LIN {X 0,Y 260.818,Z 776.411,A -85,B 0,C 180,E1 -18784.461,E2 -18784.461} C_VEL
LIN {X 0,Y 257.171,Z 786.546,A -85,B 0,C 180,E1 -18786.657,E2 -18786.657} C_VEL
LIN {X 0,Y 253.713,Z 796.339,A -85,B 0,C 180,E1 -18789.319,E2 -18789.319} C_VEL
LIN {X 0,Y 251.091,Z 804.227,A -85,B 0,C 180,E1 -18792.069,E2 -18792.069} C_VEL
LIN {X 0,Y 249.103,Z 811.376,A -85,B 0,C 180,E1 -18795.292,E2 -18795.292} C_VEL
LIN {X 0,Y 248.205,Z 815.496,A -85,B 0,C 180,E1 -18797.74,E2 -18797.74} C_VEL
LIN {X 0,Y 247.91,Z 818.682,A -85,B 0,C 180,E1 -18800.208,E2 -18800.208} C_VEL
LIN {X 0,Y 248.066,Z 820.87,A -85,B 0,C 180,E1 -18802.569,E2 -18802.569} C_VEL
LIN {X 0,Y 248.583,Z 822.288,A -85,B 0,C 180,E1 -18805.135,E2 -18805.135} C_VEL
LIN {X 0,Y 248.948,Z 822.609,A -85,B 0,C 180,E1 -18806.764,E2 -18806.764} C_VEL
LIN {X 0,Y 249.746,Z 822.308,A -85,B 0,C 180,E1 -18809.396,E2 -18809.396} C_VEL
LIN {X 0,Y 249.833,Z 822.747,A -85,B 0,C 180,E1 -18810.001,E2 -18810.001} C_VEL
LIN {X 0,Y 249.274,Z 823.471,A -85,B 0,C 180,E1 -18811.617,E2 -18811.617} C_VEL
LIN {X 0,Y 248.833,Z 823.769,A -85,B 0,C 180,E1 -18813.239,E2 -18813.239} C_VEL
LIN {X 0,Y 248.449,Z 823.635,A -85,B 0,C 180,E1 -18814.869,E2 -18814.869} C_VEL
LIN {X 0,Y 247.848,Z 822.097,A -85,B 0,C 180,E1 -18818.152,E2 -18818.152} C_VEL
LIN {X 0,Y 247.929,Z 818.939,A -85,B 0,C 180,E1 -18821.446,E2 -18821.446} C_VEL
LIN {X 0,Y 248.989,Z 814.223,A -85,B 0,C 180,E1 -18824.717,E2 -18824.717} C_VEL
LIN {X 0,Y 250.924,Z 807.901,A -85,B 0,C 180,E1 -18827.945,E2 -18827.945} C_VEL
LIN {X 0,Y 253.773,Z 800.921,A -85,B 0,C 180,E1 -18830.678,E2 -18830.678} C_VEL
LIN {X 0,Y 257.433,Z 792.435,A -85,B 0,C 180,E1 -18833.32,E2 -18833.32} C_VEL
LIN {X 0,Y 261.134,Z 783.798,A -85,B 0,C 180,E1 -18835.507,E2 -18835.507} C_VEL
LIN {X 0,Y 266.249,Z 771.804,A -85,B 0,C 180,E1 -18837.94,E2 -18837.94} C_VEL
LIN {X 0,Y 271.015,Z 760.595,A -85,B 0,C 180,E1 -18839.733,E2 -18839.733} C_VEL
LIN {X 0,Y 276.161,Z 747.47,A -85,B 0,C 180,E1 -18841.447,E2 -18841.447} C_VEL
LIN {X 0,Y 281.786,Z 731.575,A -85,B 0,C 180,E1 -18843.065,E2 -18843.065} C_VEL
LIN {X 0,Y 286.827,Z 715.559,A -85,B 0,C 180,E1 -18844.303,E2 -18844.303} C_VEL
LIN {X 0,Y 291.383,Z 697.801,A -85,B 0,C 180,E1 -18845.372,E2 -18845.372} C_VEL
LIN {X 0,Y 293.955,Z 682.068,A -85,B 0,C 180,E1 -18846.336,E2 -18846.336} C_VEL
LIN {X 0,Y 295.389,Z 669.131,A -85,B 0,C 180,E1 -18847.143,E2 -18847.143} C_VEL
LIN {X 0,Y 296.48,Z 656.031,A -85,B 0,C 180,E1 -18848.176,E2 -18848.176} C_VEL
LIN {X 0,Y 297.436,Z 642.354,A -85,B 0,C 180,E1 -18849.532,E2 -18849.532} C_VEL
LIN {X 0,Y 298.39,Z 628.951,A -85,B 0,C 180,E1 -18851.163,E2 -18851.163} C_VEL
LIN {X 0,Y 298.557,Z 626.848,A -85,B 0,C 180,E1 -18851.458,E2 -18851.458} C_VEL
LIN {X 0,Y 297.497,Z 623.568,A -85,B 0,C 180,E1 -18853.968,E2 -18853.968} C_VEL
LIN {X 0,Y 297.34,Z 623.4,A -85,B 0,C 180,E1 -18856.728,E2 -18856.728} C_VEL
LIN {X 0,Y 297.736,Z 623.726,A -85,B 0,C 180,E1 -18857.889,E2 -18857.889} C_VEL
LIN {X 0,Y 299.108,Z 626.961,A -85,B 0,C 180,E1 -18860.284,E2 -18860.284} C_VEL
LIN {X 0,Y 300.421,Z 629.677,A -85,B 0,C 180,E1 -18861.677,E2 -18861.677} C_VEL
LIN {X 0,Y 301.995,Z 633.313,A -85,B 0,C 180,E1 -18863.024,E2 -18863.024} C_VEL
LIN {X 0,Y 299.757,Z 652.581,A -85,B 0,C 180,E1 -18864.07,E2 -18864.07} C_VEL
LIN {X 0,Y 297.384,Z 666.673,A -85,B 0,C 180,E1 -18865.096,E2 -18865.096} C_VEL
LIN {X 0,Y 294.073,Z 681.241,A -85,B 0,C 180,E1 -18866.45,E2 -18866.45} C_VEL
LIN {X 0,Y 290.628,Z 693.312,A -85,B 0,C 180,E1 -18867.858,E2 -18867.858} C_VEL
LIN {X 0,Y 286.356,Z 705.963,A -85,B 0,C 180,E1 -18869.684,E2 -18869.684} C_VEL
LIN {X 0,Y 282.513,Z 715.583,A -85,B 0,C 180,E1 -18871.387,E2 -18871.387} C_VEL
LIN {X 0,Y 278.319,Z 724.834,A -85,B 0,C 180,E1 -18873.37,E2 -18873.37} C_VEL
LIN {X 0,Y 273.752,Z 733.753,A -85,B 0,C 180,E1 -18875.746,E2 -18875.746} C_VEL
LIN {X 0,Y 268.985,Z 741.99,A -85,B 0,C 180,E1 -18878.543,E2 -18878.543} C_VEL
LIN {X 0,Y 264.72,Z 748.465,A -85,B 0,C 180,E1 -18881.422,E2 -18881.422} C_VEL
LIN {X 0,Y 260.983,Z 753.365,A -85,B 0,C 180,E1 -18884.377,E2 -18884.377} C_VEL
LIN {X 0,Y 257.686,Z 756.898,A -85,B 0,C 180,E1 -18887.397,E2 -18887.397} C_VEL
LIN {X 0,Y 255.181,Z 759.04,A -85,B 0,C 180,E1 -18890.488,E2 -18890.488} C_VEL
LIN {X 0,Y 253.034,Z 760.013,A -85,B 0,C 180,E1 -18893.621,E2 -18893.621} C_VEL
LIN {X 0,Y 251.501,Z 759.716,A -85,B 0,C 180,E1 -18896.795,E2 -18896.795} C_VEL
LIN {X 0,Y 250.423,Z 758.19,A -85,B 0,C 180,E1 -18899.999,E2 -18899.999} C_VEL
LIN {X 0,Y 249.712,Z 755.413,A -85,B 0,C 180,E1 -18903.226,E2 -18903.226} C_VEL
LIN {X 0,Y 249.459,Z 751.304,A -85,B 0,C 180,E1 -18906.47,E2 -18906.47} C_VEL
LIN {X 0,Y 249.698,Z 745.77,A -85,B 0,C 180,E1 -18909.722,E2 -18909.722} C_VEL
LIN {X 0,Y 250.129,Z 738.659,A -85,B 0,C 180,E1 -18912.989,E2 -18912.989} C_VEL
LIN {X 0,Y 250.911,Z 730.916,A -85,B 0,C 180,E1 -18915.848,E2 -18915.848} C_VEL
LIN {X 0,Y 252.025,Z 721.082,A -85,B 0,C 180,E1 -18918.823,E2 -18918.823} C_VEL
LIN {X 0,Y 253.137,Z 711.784,A -85,B 0,C 180,E1 -18921.156,E2 -18921.156} C_VEL
LIN {X 0,Y 254.594,Z 700.217,A -85,B 0,C 180,E1 -18923.594,E2 -18923.594} C_VEL
LIN {X 0,Y 256.131,Z 687.264,A -85,B 0,C 180,E1 -18925.84,E2 -18925.84} C_VEL
LIN {X 0,Y 257.565,Z 674.72,A -85,B 0,C 180,E1 -18927.636,E2 -18927.636} C_VEL
LIN {X 0,Y 258.908,Z 660.999,A -85,B 0,C 180,E1 -18929.248,E2 -18929.248} C_VEL
LIN {X 0,Y 260.031,Z 646.822,A -85,B 0,C 180,E1 -18930.585,E2 -18930.585} C_VEL
LIN {X 0,Y 261.021,Z 631.089,A -85,B 0,C 180,E1 -18931.727,E2 -18931.727} C_VEL
LIN {X 0,Y 261.687,Z 615.325,A -85,B 0,C 180,E1 -18932.546,E2 -18932.546} C_VEL
LIN {X 0,Y 261.742,Z 605.267,A -85,B 0,C 180,E1 -18932.982,E2 -18932.982} C_VEL
LIN {X 0,Y 249.083,Z 569.455,A -85,B 0,C 180,E1 -18935.438,E2 -18935.438} C_VEL
LIN {X 0,Y 249.029,Z 569.466,A -85,B 0,C 180,E1 -18938.379,E2 -18938.379} C_VEL
LIN {X 0,Y 249.01,Z 569.466,A -85,B 0,C 180,E1 -18942.791,E2 -18942.791} C_VEL
LIN {X 0,Y 249.02,Z 569.462,A -85,B 0,C 180,E1 -18947.362,E2 -18947.362} C_VEL
LIN {X 0,Y 249.04,Z 569.461,A -85,B 0,C 180,E1 -18951.621,E2 -18951.621} C_VEL
LIN {X 0,Y 249.061,Z 569.458,A -85,B 0,C 180,E1 -18955.641,E2 -18955.641} C_VEL
LIN {X 0,Y 249.047,Z 569.459,A -85,B 0,C 180,E1 -18959.471,E2 -18959.471} C_VEL
LIN {X 0,Y 249.071,Z 569.458,A -85,B 0,C 180,E1 -18963.161,E2 -18963.161} C_VEL
LIN {X 0,Y 249.079,Z 569.458,A -85,B 0,C 180,E1 -18966.732,E2 -18966.732} C_VEL
LIN {X 0,Y 249.11,Z 569.453,A -85,B 0,C 180,E1 -18970.211,E2 -18970.211} C_VEL
LIN {X 0,Y 249.241,Z 569.435,A -85,B 0,C 180,E1 -18973.621,E2 -18973.621} C_VEL
LIN {X 0,Y 249.252,Z 569.436,A -85,B 0,C 180,E1 -18978.616,E2 -18978.616} C_VEL
LIN {X 0,Y 249.483,Z 569.405,A -85,B 0,C 180,E1 -18981.902,E2 -18981.902} C_VEL
LIN {X 0,Y 249.435,Z 569.413,A -85,B 0,C 180,E1 -18986.769,E2 -18986.769} C_VEL
LIN {X 0,Y 249.727,Z 569.375,A -85,B 0,C 180,E1 -18989.999,E2 -18989.999} C_VEL
LIN {X 0,Y 249.435,Z 569.413,A -85,B 0,C 180,E1 -18993.229,E2 -18993.229} C_VEL
LIN {X 0,Y 249.481,Z 569.406,A -85,B 0,C 180,E1 -18998.096,E2 -18998.096} C_VEL
LIN {X 0,Y 249.251,Z 569.436,A -85,B 0,C 180,E1 -19001.383,E2 -19001.383} C_VEL
LIN {X 0,Y 249.238,Z 569.436,A -85,B 0,C 180,E1 -19006.377,E2 -19006.377} C_VEL
LIN {X 0,Y 249.123,Z 569.452,A -85,B 0,C 180,E1 -19011.417,E2 -19011.417} C_VEL
LIN {X 0,Y 249.127,Z 569.454,A -85,B 0,C 180,E1 -19015.482,E2 -19015.482} C_VEL
LIN {X 0,Y 249.076,Z 569.455,A -85,B 0,C 180,E1 -19018.992,E2 -19018.992} C_VEL
LIN {X 0,Y 249.032,Z 569.462,A -85,B 0,C 180,E1 -19022.424,E2 -19022.424} C_VEL
LIN {X 0,Y 249.071,Z 569.458,A -85,B 0,C 180,E1 -19026.337,E2 -19026.337} C_VEL
LIN {X 0,Y 249.041,Z 569.462,A -85,B 0,C 180,E1 -19030.47,E2 -19030.47} C_VEL
LIN {X 0,Y 249.055,Z 569.46,A -85,B 0,C 180,E1 -19034.866,E2 -19034.866} C_VEL
LIN {X 0,Y 249.139,Z 569.567,A -85,B 0,C 180,E1 -19036.965,E2 -19036.965} C_VEL
LIN {X 0,Y 260.84,Z 601.69,A -85,B 0,C 180,E1 -19039.114,E2 -19039.114} C_VEL
LIN {X 0,Y 259.994,Z 636.39,A -85,B 0,C 180,E1 -19040.501,E2 -19040.501} C_VEL
LIN {X 0,Y 259.352,Z 649.977,A -85,B 0,C 180,E1 -19041.322,E2 -19041.322} C_VEL
LIN {X 0,Y 258.459,Z 663.068,A -85,B 0,C 180,E1 -19042.395,E2 -19042.395} C_VEL
LIN {X 0,Y 257.324,Z 676.378,A -85,B 0,C 180,E1 -19043.8,E2 -19043.8} C_VEL
LIN {X 0,Y 255.939,Z 689.02,A -85,B 0,C 180,E1 -19045.464,E2 -19045.464} C_VEL
LIN {X 0,Y 254.583,Z 701.023,A -85,B 0,C 180,E1 -19047.432,E2 -19047.432} C_VEL
LIN {X 0,Y 253.176,Z 712.056,A -85,B 0,C 180,E1 -19049.643,E2 -19049.643} C_VEL
LIN {X 0,Y 251.937,Z 722.278,A -85,B 0,C 180,E1 -19052.145,E2 -19052.145} C_VEL
LIN {X 0,Y 250.922,Z 730.795,A -85,B 0,C 180,E1 -19054.715,E2 -19054.715} C_VEL
LIN {X 0,Y 250.063,Z 738.633,A -85,B 0,C 180,E1 -19057.652,E2 -19057.652} C_VEL
LIN {X 0,Y 249.542,Z 744.184,A -85,B 0,C 180,E1 -19060.248,E2 -19060.248} C_VEL
LIN {X 0,Y 249.323,Z 749.439,A -85,B 0,C 180,E1 -19063.412,E2 -19063.412} C_VEL
LIN {X 0,Y 249.327,Z 751.809,A -85,B 0,C 180,E1 -19065.305,E2 -19065.305} C_VEL
LIN {X 0,Y 249.763,Z 754.792,A -85,B 0,C 180,E1 -19068.641,E2 -19068.641} C_VEL
LIN {X 0,Y 250.168,Z 755.714,A -85,B 0,C 180,E1 -19070.297,E2 -19070.297} C_VEL
LIN {X 0,Y 250.609,Z 756.259,A -85,B 0,C 180,E1 -19071.94,E2 -19071.94} C_VEL
LIN {X 0,Y 251.976,Z 756.187,A -85,B 0,C 180,E1 -19075.201,E2 -19075.201} C_VEL
LIN {X 0,Y 253.827,Z 754.677,A -85,B 0,C 180,E1 -19078.414,E2 -19078.414} C_VEL
LIN {X 0,Y 256.246,Z 751.663,A -85,B 0,C 180,E1 -19081.572,E2 -19081.572} C_VEL
LIN {X 0,Y 258.413,Z 748.364,A -85,B 0,C 180,E1 -19083.899,E2 -19083.899} C_VEL
LIN {X 0,Y 260.8,Z 744.134,A -85,B 0,C 180,E1 -19086.189,E2 -19086.189} C_VEL
LIN {X 0,Y 263.99,Z 737.967,A -85,B 0,C 180,E1 -19088.756,E2 -19088.756} C_VEL
LIN {X 0,Y 267.696,Z 729.874,A -85,B 0,C 180,E1 -19091.357,E2 -19091.357} C_VEL
LIN {X 0,Y 271.027,Z 721.524,A -85,B 0,C 180,E1 -19093.497,E2 -19093.497} C_VEL
LIN {X 0,Y 274.007,Z 713.118,A -85,B 0,C 180,E1 -19095.243,E2 -19095.243} C_VEL
LIN {X 0,Y 277.39,Z 702.417,A -85,B 0,C 180,E1 -19097.066,E2 -19097.066} C_VEL
LIN {X 0,Y 278.319,Z 697.956,A -85,B 0,C 180,E1 -19097.845,E2 -19097.845} C_VEL
LIN {X 0,Y 278.464,Z 690.905,A -85,B 0,C 180,E1 -19099.284,E2 -19099.284} C_VEL
LIN {X 0,Y 278.414,Z 683.478,A -85,B 0,C 180,E1 -19100.624,E2 -19100.624} C_VEL
LIN {X 0,Y 278.977,Z 678.441,A -85,B 0,C 180,E1 -19101.237,E2 -19101.237} C_VEL
LIN {X 0,Y 281.141,Z 664.751,A -85,B 0,C 180,E1 -19102.399,E2 -19102.399} C_VEL
LIN {X 0,Y 282.696,Z 651.495,A -85,B 0,C 180,E1 -19103.228,E2 -19103.228} C_VEL
LIN {X 0,Y 284.503,Z 629.994,A -85,B 0,C 180,E1 -19104.228,E2 -19104.228} C_VEL
LIN {X 0,Y 284.814,Z 626.374,A -85,B 0,C 180,E1 -19104.395,E2 -19104.395} C_VEL
LIN {X 0,Y 281.706,Z 620.21,A -85,B 0,C 180,E1 -19106.089,E2 -19106.089} C_VEL
LIN {X 0,Y 278.294,Z 614.051,A -85,B 0,C 180,E1 -19108.276,E2 -19108.276} C_VEL
LIN {X 0,Y 275.873,Z 610.077,A -85,B 0,C 180,E1 -19110.204,E2 -19110.204} C_VEL
LIN {X 0,Y 273.888,Z 607.248,A -85,B 0,C 180,E1 -19112.202,E2 -19112.202} C_VEL
LIN {X 0,Y 273.43,Z 605.988,A -85,B 0,C 180,E1 -19112.906,E2 -19112.906} C_VEL
LIN {X 0,Y 271.454,Z 604.131,A -85,B 0,C 180,E1 -19116.623,E2 -19116.623} C_VEL
LIN {X 0,Y 271.349,Z 604.083,A -85,B 0,C 180,E1 -19119.623,E2 -19119.623} C_VEL
LIN {X 0,Y 273.172,Z 605.872,A -85,B 0,C 180,E1 -19123.492,E2 -19123.492} C_VEL
LIN {X 0,Y 274.768,Z 609.373,A -85,B 0,C 180,E1 -19125.606,E2 -19125.606} C_VEL
LIN {X 0,Y 276.198,Z 618.214,A -85,B 0,C 180,E1 -19127.826,E2 -19127.826} C_VEL
LIN {X 0,Y 277.197,Z 625.336,A -85,B 0,C 180,E1 -19129.213,E2 -19129.213} C_VEL
LIN {X 0,Y 277.67,Z 641.94,A -85,B 0,C 180,E1 -19131.142,E2 -19131.142} C_VEL
LIN {X 0,Y 277.968,Z 659.419,A -85,B 0,C 180,E1 -19132.848,E2 -19132.848} C_VEL
LIN {X 0,Y 277.908,Z 669.287,A -85,B 0,C 180,E1 -19133.643,E2 -19133.643} C_VEL
LIN {X 0,Y 277.1,Z 695.717,A -85,B 0,C 180,E1 -19135.458,E2 -19135.458} C_VEL
LIN {X 0,Y 274.741,Z 710.764,A -85,B 0,C 180,E1 -19136.209,E2 -19136.209} C_VEL
LIN {X 0,Y 271.163,Z 726.585,A -85,B 0,C 180,E1 -19137.247,E2 -19137.247} C_VEL
LIN {X 0,Y 267.245,Z 740.848,A -85,B 0,C 180,E1 -19138.489,E2 -19138.489} C_VEL
LIN {X 0,Y 263.128,Z 753.709,A -85,B 0,C 180,E1 -19139.948,E2 -19139.948} C_VEL
LIN {X 0,Y 258.602,Z 766.608,A -85,B 0,C 180,E1 -19141.824,E2 -19141.824} C_VEL
LIN {X 0,Y 254.486,Z 777.288,A -85,B 0,C 180,E1 -19143.778,E2 -19143.778} C_VEL
LIN {X 0,Y 250.707,Z 787.047,A -85,B 0,C 180,E1 -19146.018,E2 -19146.018} C_VEL
LIN {X 0,Y 247.539,Z 795.209,A -85,B 0,C 180,E1 -19148.342,E2 -19148.342} C_VEL
LIN {X 0,Y 245.009,Z 802.018,A -85,B 0,C 180,E1 -19150.74,E2 -19150.74} C_VEL
LIN {X 0,Y 243.138,Z 807.696,A -85,B 0,C 180,E1 -19153.2,E2 -19153.2} C_VEL
LIN {X 0,Y 241.798,Z 812.291,A -85,B 0,C 180,E1 -19155.698,E2 -19155.698} C_VEL
LIN {X 0,Y 241.029,Z 815.929,A -85,B 0,C 180,E1 -19158.224,E2 -19158.224} C_VEL
LIN {X 0,Y 240.843,Z 817.86,A -85,B 0,C 180,E1 -19159.917,E2 -19159.917} C_VEL
LIN {X 0,Y 241.001,Z 820.011,A -85,B 0,C 180,E1 -19162.528,E2 -19162.528} C_VEL
LIN {X 0,Y 241.51,Z 821.165,A -85,B 0,C 180,E1 -19164.993,E2 -19164.993} C_VEL
LIN {X 0,Y 241.901,Z 821.421,A -85,B 0,C 180,E1 -19166.67,E2 -19166.67} C_VEL
LIN {X 0,Y 242.834,Z 820.928,A -85,B 0,C 180,E1 -19169.586,E2 -19169.586} C_VEL
LIN {X 0,Y 242.891,Z 821.272,A -85,B 0,C 180,E1 -19170.001,E2 -19170.001} C_VEL
LIN {X 0,Y 242.288,Z 822.074,A -85,B 0,C 180,E1 -19171.663,E2 -19171.663} C_VEL
LIN {X 0,Y 241.831,Z 822.454,A -85,B 0,C 180,E1 -19173.333,E2 -19173.333} C_VEL
LIN {X 0,Y 241.389,Z 822.399,A -85,B 0,C 180,E1 -19175.012,E2 -19175.012} C_VEL
LIN {X 0,Y 240.782,Z 821.056,A -85,B 0,C 180,E1 -19178.393,E2 -19178.393} C_VEL
LIN {X 0,Y 240.904,Z 818.16,A -85,B 0,C 180,E1 -19181.784,E2 -19181.784} C_VEL
LIN {X 0,Y 242.053,Z 813.751,A -85,B 0,C 180,E1 -19185.149,E2 -19185.149} C_VEL
LIN {X 0,Y 244.167,Z 807.726,A -85,B 0,C 180,E1 -19188.46,E2 -19188.46} C_VEL
LIN {X 0,Y 247.605,Z 800.027,A -85,B 0,C 180,E1 -19191.654,E2 -19191.654} C_VEL
LIN {X 0,Y 251.513,Z 791.74,A -85,B 0,C 180,E1 -19194.341,E2 -19194.341} C_VEL
LIN {X 0,Y 256.308,Z 781.801,A -85,B 0,C 180,E1 -19196.901,E2 -19196.901} C_VEL
LIN {X 0,Y 260.94,Z 771.732,A -85,B 0,C 180,E1 -19199,E2 -19199} C_VEL
LIN {X 0,Y 266.366,Z 759.831,A -85,B 0,C 180,E1 -19200.965,E2 -19200.965} C_VEL
LIN {X 0,Y 271.822,Z 746.995,A -85,B 0,C 180,E1 -19202.666,E2 -19202.666} C_VEL
LIN {X 0,Y 277.161,Z 733.226,A -85,B 0,C 180,E1 -19204.128,E2 -19204.128} C_VEL
LIN {X 0,Y 282.378,Z 718.186,A -85,B 0,C 180,E1 -19205.357,E2 -19205.357} C_VEL
LIN {X 0,Y 287.426,Z 700.862,A -85,B 0,C 180,E1 -19206.476,E2 -19206.476} C_VEL
LIN {X 0,Y 289.357,Z 692.202,A -85,B 0,C 180,E1 -19207.007,E2 -19207.007} C_VEL
LIN {X 0,Y 292.418,Z 673.252,A -85,B 0,C 180,E1 -19208.206,E2 -19208.206} C_VEL
LIN {X 0,Y 293.903,Z 659.145,A -85,B 0,C 180,E1 -19209.311,E2 -19209.311} C_VEL
LIN {X 0,Y 295.183,Z 645.582,A -85,B 0,C 180,E1 -19210.671,E2 -19210.671} C_VEL
LIN {X 0,Y 296.464,Z 633.107,A -85,B 0,C 180,E1 -19212.209,E2 -19212.209} C_VEL
LIN {X 0,Y 295.886,Z 630.41,A -85,B 0,C 180,E1 -19214.26,E2 -19214.26} C_VEL
LIN {X 0,Y 295.773,Z 630.322,A -85,B 0,C 180,E1 -19216.442,E2 -19216.442} C_VEL
LIN {X 0,Y 296.19,Z 630.746,A -85,B 0,C 180,E1 -19217.805,E2 -19217.805} C_VEL
LIN {X 0,Y 297.401,Z 633.722,A -85,B 0,C 180,E1 -19220.053,E2 -19220.053} C_VEL
LIN {X 0,Y 298.922,Z 637.403,A -85,B 0,C 180,E1 -19221.762,E2 -19221.762} C_VEL
LIN {X 0,Y 299.134,Z 637.956,A -85,B 0,C 180,E1 -19221.957,E2 -19221.957} C_VEL
LIN {X 0,Y 296.908,Z 654.624,A -85,B 0,C 180,E1 -19222.885,E2 -19222.885} C_VEL
LIN {X 0,Y 294.192,Z 669.261,A -85,B 0,C 180,E1 -19223.965,E2 -19223.965} C_VEL
LIN {X 0,Y 290.885,Z 682.656,A -85,B 0,C 180,E1 -19225.233,E2 -19225.233} C_VEL
LIN {X 0,Y 286.873,Z 695.629,A -85,B 0,C 180,E1 -19226.759,E2 -19226.759} C_VEL
LIN {X 0,Y 283.105,Z 706.05,A -85,B 0,C 180,E1 -19228.265,E2 -19228.265} C_VEL
LIN {X 0,Y 278.602,Z 716.67,A -85,B 0,C 180,E1 -19230.118,E2 -19230.118} C_VEL
LIN {X 0,Y 274.16,Z 725.948,A -85,B 0,C 180,E1 -19232.106,E2 -19232.106} C_VEL
LIN {X 0,Y 269.244,Z 734.861,A -85,B 0,C 180,E1 -19234.488,E2 -19234.488} C_VEL
LIN {X 0,Y 265.365,Z 741.267,A -85,B 0,C 180,E1 -19236.592,E2 -19236.592} C_VEL
LIN {X 0,Y 260.58,Z 748.126,A -85,B 0,C 180,E1 -19239.474,E2 -19239.474} C_VEL
LIN {X 0,Y 256.362,Z 753.466,A -85,B 0,C 180,E1 -19242.448,E2 -19242.448} C_VEL
LIN {X 0,Y 252.686,Z 757.327,A -85,B 0,C 180,E1 -19245.503,E2 -19245.503} C_VEL
LIN {X 0,Y 249.555,Z 759.921,A -85,B 0,C 180,E1 -19248.63,E2 -19248.63} C_VEL
LIN {X 0,Y 247.198,Z 761.179,A -85,B 0,C 180,E1 -19251.827,E2 -19251.827} C_VEL
LIN {X 0,Y 245.257,Z 761.248,A -85,B 0,C 180,E1 -19255.068,E2 -19255.068} C_VEL
LIN {X 0,Y 243.85,Z 760.091,A -85,B 0,C 180,E1 -19258.348,E2 -19258.348} C_VEL
LIN {X 0,Y 242.964,Z 757.682,A -85,B 0,C 180,E1 -19261.657,E2 -19261.657} C_VEL
LIN {X 0,Y 242.381,Z 754.003,A -85,B 0,C 180,E1 -19264.99,E2 -19264.99} C_VEL
LIN {X 0,Y 242.508,Z 748.915,A -85,B 0,C 180,E1 -19268.331,E2 -19268.331} C_VEL
LIN {X 0,Y 242.83,Z 742.321,A -85,B 0,C 180,E1 -19271.688,E2 -19271.688} C_VEL
LIN {X 0,Y 243.389,Z 735.105,A -85,B 0,C 180,E1 -19274.634,E2 -19274.634} C_VEL
LIN {X 0,Y 244.398,Z 726.349,A -85,B 0,C 180,E1 -19277.573,E2 -19277.573} C_VEL
LIN {X 0,Y 245.482,Z 717.339,A -85,B 0,C 180,E1 -19280.093,E2 -19280.093} C_VEL
LIN {X 0,Y 246.983,Z 705.659,A -85,B 0,C 180,E1 -19282.811,E2 -19282.811} C_VEL
LIN {X 0,Y 248.509,Z 693.257,A -85,B 0,C 180,E1 -19285.178,E2 -19285.178} C_VEL
LIN {X 0,Y 249.99,Z 680.571,A -85,B 0,C 180,E1 -19287.182,E2 -19287.182} C_VEL
LIN {X 0,Y 251.33,Z 667.895,A -85,B 0,C 180,E1 -19288.839,E2 -19288.839} C_VEL
LIN {X 0,Y 252.58,Z 654.444,A -85,B 0,C 180,E1 -19290.274,E2 -19290.274} C_VEL
LIN {X 0,Y 253.68,Z 639.263,A -85,B 0,C 180,E1 -19291.555,E2 -19291.555} C_VEL
LIN {X 0,Y 254.485,Z 623.91,A -85,B 0,C 180,E1 -19292.522,E2 -19292.522} C_VEL
LIN {X 0,Y 254.934,Z 606.988,A -85,B 0,C 180,E1 -19293.292,E2 -19293.292} C_VEL
LIN {X 0,Y 242.055,Z 570.333,A -85,B 0,C 180,E1 -19295.933,E2 -19295.933} C_VEL
LIN {X 0,Y 241.958,Z 570.344,A -85,B 0,C 180,E1 -19299.718,E2 -19299.718} C_VEL
LIN {X 0,Y 241.931,Z 570.35,A -85,B 0,C 180,E1 -19304.201,E2 -19304.201} C_VEL
LIN {X 0,Y 241.946,Z 570.346,A -85,B 0,C 180,E1 -19308.078,E2 -19308.078} C_VEL
LIN {X 0,Y 242.003,Z 570.341,A -85,B 0,C 180,E1 -19312.42,E2 -19312.42} C_VEL
LIN {X 0,Y 241.991,Z 570.341,A -85,B 0,C 180,E1 -19316.508,E2 -19316.508} C_VEL
LIN {X 0,Y 242.013,Z 570.34,A -85,B 0,C 180,E1 -19320.596,E2 -19320.596} C_VEL
LIN {X 0,Y 242.067,Z 570.33,A -85,B 0,C 180,E1 -19324.182,E2 -19324.182} C_VEL
LIN {X 0,Y 242.052,Z 570.331,A -85,B 0,C 180,E1 -19328.296,E2 -19328.296} C_VEL
LIN {X 0,Y 242.162,Z 570.318,A -85,B 0,C 180,E1 -19333.277,E2 -19333.277} C_VEL
LIN {X 0,Y 242.185,Z 570.315,A -85,B 0,C 180,E1 -19338.279,E2 -19338.279} C_VEL
LIN {X 0,Y 242.434,Z 570.284,A -85,B 0,C 180,E1 -19341.665,E2 -19341.665} C_VEL
LIN {X 0,Y 242.26,Z 570.307,A -85,B 0,C 180,E1 -19345.006,E2 -19345.006} C_VEL
LIN {X 0,Y 242.635,Z 570.259,A -85,B 0,C 180,E1 -19348.339,E2 -19348.339} C_VEL
LIN {X 0,Y 242.635,Z 570.258,A -85,B 0,C 180,E1 -19351.659,E2 -19351.659} C_VEL
LIN {X 0,Y 242.431,Z 570.285,A -85,B 0,C 180,E1 -19356.658,E2 -19356.658} C_VEL
LIN {X 0,Y 242.343,Z 570.294,A -85,B 0,C 180,E1 -19360.02,E2 -19360.02} C_VEL
LIN {X 0,Y 242.164,Z 570.319,A -85,B 0,C 180,E1 -19365.14,E2 -19365.14} C_VEL
LIN {X 0,Y 242.076,Z 570.328,A -85,B 0,C 180,E1 -19368.623,E2 -19368.623} C_VEL
LIN {X 0,Y 242.046,Z 570.332,A -85,B 0,C 180,E1 -19372.176,E2 -19372.176} C_VEL
LIN {X 0,Y 242.062,Z 570.333,A -85,B 0,C 180,E1 -19375.837,E2 -19375.837} C_VEL
LIN {X 0,Y 242.025,Z 570.336,A -85,B 0,C 180,E1 -19379.58,E2 -19379.58} C_VEL
LIN {X 0,Y 241.987,Z 570.342,A -85,B 0,C 180,E1 -19383.49,E2 -19383.49} C_VEL
LIN {X 0,Y 242.008,Z 570.34,A -85,B 0,C 180,E1 -19387.577,E2 -19387.577} C_VEL
LIN {X 0,Y 241.975,Z 570.345,A -85,B 0,C 180,E1 -19391.913,E2 -19391.913} C_VEL
LIN {X 0,Y 242.087,Z 570.525,A -85,B 0,C 180,E1 -19396.472,E2 -19396.472} C_VEL
LIN {X 0,Y 254.003,Z 603.298,A -85,B 0,C 180,E1 -19398.732,E2 -19398.732} C_VEL
LIN {X 0,Y 253.093,Z 637.837,A -85,B 0,C 180,E1 -19400.158,E2 -19400.158} C_VEL
LIN {X 0,Y 252.438,Z 651.317,A -85,B 0,C 180,E1 -19401.004,E2 -19401.004} C_VEL
LIN {X 0,Y 251.419,Z 665.103,A -85,B 0,C 180,E1 -19402.178,E2 -19402.178} C_VEL
LIN {X 0,Y 250.284,Z 678.179,A -85,B 0,C 180,E1 -19403.617,E2 -19403.617} C_VEL
LIN {X 0,Y 248.842,Z 690.713,A -85,B 0,C 180,E1 -19405.335,E2 -19405.335} C_VEL
LIN {X 0,Y 247.513,Z 702.521,A -85,B 0,C 180,E1 -19407.352,E2 -19407.352} C_VEL
LIN {X 0,Y 246.116,Z 713.121,A -85,B 0,C 180,E1 -19409.546,E2 -19409.546} C_VEL
LIN {X 0,Y 244.783,Z 723.601,A -85,B 0,C 180,E1 -19412.19,E2 -19412.19} C_VEL
LIN {X 0,Y 243.751,Z 732.072,A -85,B 0,C 180,E1 -19414.832,E2 -19414.832} C_VEL
LIN {X 0,Y 242.904,Z 740.029,A -85,B 0,C 180,E1 -19417.907,E2 -19417.907} C_VEL
LIN {X 0,Y 242.442,Z 745.452,A -85,B 0,C 180,E1 -19420.528,E2 -19420.528} C_VEL
LIN {X 0,Y 242.257,Z 749.847,A -85,B 0,C 180,E1 -19423.202,E2 -19423.202} C_VEL
LIN {X 0,Y 242.415,Z 753.962,A -85,B 0,C 180,E1 -19426.59,E2 -19426.59} C_VEL
LIN {X 0,Y 243.056,Z 756.504,A -85,B 0,C 180,E1 -19430.01,E2 -19430.01} C_VEL
LIN {X 0,Y 244.137,Z 757.575,A -85,B 0,C 180,E1 -19433.389,E2 -19433.389} C_VEL
LIN {X 0,Y 245.781,Z 757.179,A -85,B 0,C 180,E1 -19436.722,E2 -19436.722} C_VEL
LIN {X 0,Y 247.973,Z 755.275,A -85,B 0,C 180,E1 -19440.001,E2 -19440.001} C_VEL
LIN {X 0,Y 250.741,Z 751.879,A -85,B 0,C 180,E1 -19443.214,E2 -19443.214} C_VEL
LIN {X 0,Y 253.177,Z 748.26,A -85,B 0,C 180,E1 -19445.576,E2 -19445.576} C_VEL
LIN {X 0,Y 255.891,Z 743.699,A -85,B 0,C 180,E1 -19447.894,E2 -19447.894} C_VEL
LIN {X 0,Y 259.511,Z 736.985,A -85,B 0,C 180,E1 -19450.534,E2 -19450.534} C_VEL
LIN {X 0,Y 262.931,Z 729.819,A -85,B 0,C 180,E1 -19452.74,E2 -19452.74} C_VEL
LIN {X 0,Y 266.517,Z 721.249,A -85,B 0,C 180,E1 -19454.899,E2 -19454.899} C_VEL
LIN {X 0,Y 269.769,Z 712.607,A -85,B 0,C 180,E1 -19456.653,E2 -19456.653} C_VEL
LIN {X 0,Y 273.4,Z 701.083,A -85,B 0,C 180,E1 -19458.549,E2 -19458.549} C_VEL
LIN {X 0,Y 276.57,Z 689.472,A -85,B 0,C 180,E1 -19460.064,E2 -19460.064} C_VEL
LIN {X 0,Y 278.977,Z 678.441,A -85,B 0,C 180,E1 -19461.237,E2 -19461.237} C_VEL
LIN {X 0,Y 279.549,Z 673.284,A -85,B 0,C 180,E1 -19461.822,E2 -19461.822} C_VEL
LIN {X 0,Y 279.259,Z 665.175,A -85,B 0,C 180,E1 -19462.995,E2 -19462.995} C_VEL
LIN {X 0,Y 278.823,Z 656.848,A -85,B 0,C 180,E1 -19464.069,E2 -19464.069} C_VEL
LIN {X 0,Y 279.009,Z 651.371,A -85,B 0,C 180,E1 -19464.494,E2 -19464.494} C_VEL
LIN {X 0,Y 280.927,Z 631.16,A -85,B 0,C 180,E1 -19465.448,E2 -19465.448} C_VEL
LIN {X 0,Y 280.95,Z 629.994,A -85,B 0,C 180,E1 -19465.537,E2 -19465.537} C_VEL
LIN {X 0,Y 277.763,Z 623.606,A -85,B 0,C 180,E1 -19467.526,E2 -19467.526} C_VEL
LIN {X 0,Y 275.403,Z 619.426,A -85,B 0,C 180,E1 -19469.266,E2 -19469.266} C_VEL
LIN {X 0,Y 273.873,Z 616.641,A -85,B 0,C 180,E1 -19470.641,E2 -19470.641} C_VEL
LIN {X 0,Y 272.015,Z 613.664,A -85,B 0,C 180,E1 -19472.712,E2 -19472.712} C_VEL
LIN {X 0,Y 271.544,Z 612.684,A -85,B 0,C 180,E1 -19473.405,E2 -19473.405} C_VEL
LIN {X 0,Y 269.961,Z 611.049,A -85,B 0,C 180,E1 -19476.782,E2 -19476.782} C_VEL
LIN {X 0,Y 269.917,Z 611.069,A -85,B 0,C 180,E1 -19479.762,E2 -19479.762} C_VEL
LIN {X 0,Y 271.577,Z 612.855,A -85,B 0,C 180,E1 -19483.391,E2 -19483.391} C_VEL
LIN {X 0,Y 272.614,Z 615.708,A -85,B 0,C 180,E1 -19485.007,E2 -19485.007} C_VEL
LIN {X 0,Y 273.574,Z 623.201,A -85,B 0,C 180,E1 -19486.919,E2 -19486.919} C_VEL
LIN {X 0,Y 274.271,Z 629.565,A -85,B 0,C 180,E1 -19488.173,E2 -19488.173} C_VEL
LIN {X 0,Y 274.361,Z 644.983,A -85,B 0,C 180,E1 -19489.996,E2 -19489.996} C_VEL
LIN {X 0,Y 274.36,Z 662.015,A -85,B 0,C 180,E1 -19491.705,E2 -19491.705} C_VEL
LIN {X 0,Y 274.075,Z 671.996,A -85,B 0,C 180,E1 -19492.523,E2 -19492.523} C_VEL
LIN {X 0,Y 272.976,Z 696.645,A -85,B 0,C 180,E1 -19494.271,E2 -19494.271} C_VEL
LIN {X 0,Y 270.19,Z 712.002,A -85,B 0,C 180,E1 -19495.094,E2 -19495.094} C_VEL
LIN {X 0,Y 266.419,Z 727.301,A -85,B 0,C 180,E1 -19496.134,E2 -19496.134} C_VEL
LIN {X 0,Y 262.337,Z 740.886,A -85,B 0,C 180,E1 -19497.376,E2 -19497.376} C_VEL
LIN {X 0,Y 257.571,Z 754.669,A -85,B 0,C 180,E1 -19499.003,E2 -19499.003} C_VEL
LIN {X 0,Y 252.843,Z 767.051,A -85,B 0,C 180,E1 -19500.895,E2 -19500.895} C_VEL
LIN {X 0,Y 248.194,Z 778.222,A -85,B 0,C 180,E1 -19503.061,E2 -19503.061} C_VEL
LIN {X 0,Y 244.273,Z 787.521,A -85,B 0,C 180,E1 -19505.344,E2 -19505.344} C_VEL
LIN {X 0,Y 240.456,Z 796.516,A -85,B 0,C 180,E1 -19508.122,E2 -19508.122} C_VEL
LIN {X 0,Y 237.569,Z 803.819,A -85,B 0,C 180,E1 -19511.011,E2 -19511.011} C_VEL
LIN {X 0,Y 235.76,Z 808.91,A -85,B 0,C 180,E1 -19513.55,E2 -19513.55} C_VEL
LIN {X 0,Y 234.211,Z 814.125,A -85,B 0,C 180,E1 -19516.995,E2 -19516.995} C_VEL
LIN {X 0,Y 233.781,Z 816.996,A -85,B 0,C 180,E1 -19519.61,E2 -19519.61} C_VEL
LIN {X 0,Y 234.012,Z 819.413,A -85,B 0,C 180,E1 -19523.101,E2 -19523.101} C_VEL
LIN {X 0,Y 234.44,Z 820.041,A -85,B 0,C 180,E1 -19524.841,E2 -19524.841} C_VEL
LIN {X 0,Y 234.852,Z 820.227,A -85,B 0,C 180,E1 -19526.57,E2 -19526.57} C_VEL
LIN {X 0,Y 235.932,Z 819.523,A -85,B 0,C 180,E1 -19529.788,E2 -19529.788} C_VEL
LIN {X 0,Y 235.322,Z 820.612,A -85,B 0,C 180,E1 -19531.712,E2 -19531.712} C_VEL
LIN {X 0,Y 234.819,Z 821.108,A -85,B 0,C 180,E1 -19533.433,E2 -19533.433} C_VEL
LIN {X 0,Y 234.331,Z 821.154,A -85,B 0,C 180,E1 -19535.163,E2 -19535.163} C_VEL
LIN {X 0,Y 233.718,Z 820.013,A -85,B 0,C 180,E1 -19538.648,E2 -19538.648} C_VEL
LIN {X 0,Y 233.902,Z 817.347,A -85,B 0,C 180,E1 -19542.143,E2 -19542.143} C_VEL
LIN {X 0,Y 235.14,Z 813.203,A -85,B 0,C 180,E1 -19545.606,E2 -19545.606} C_VEL
LIN {X 0,Y 236.567,Z 809.297,A -85,B 0,C 180,E1 -19548.07,E2 -19548.07} C_VEL
LIN {X 0,Y 239.122,Z 804.128,A -85,B 0,C 180,E1 -19550.653,E2 -19550.653} C_VEL
LIN {X 0,Y 242.721,Z 797.077,A -85,B 0,C 180,E1 -19553.462,E2 -19553.462} C_VEL
LIN {X 0,Y 247.148,Z 788.57,A -85,B 0,C 180,E1 -19556.154,E2 -19556.154} C_VEL
LIN {X 0,Y 252.39,Z 778.399,A -85,B 0,C 180,E1 -19558.709,E2 -19558.709} C_VEL
LIN {X 0,Y 257.551,Z 768.145,A -85,B 0,C 180,E1 -19560.774,E2 -19560.774} C_VEL
LIN {X 0,Y 263.929,Z 755.012,A -85,B 0,C 180,E1 -19562.859,E2 -19562.859} C_VEL
LIN {X 0,Y 270.411,Z 740.44,A -85,B 0,C 180,E1 -19564.649,E2 -19564.649} C_VEL
LIN {X 0,Y 275.616,Z 727.465,A -85,B 0,C 180,E1 -19565.909,E2 -19565.909} C_VEL
LIN {X 0,Y 281.248,Z 711.715,A -85,B 0,C 180,E1 -19567.098,E2 -19567.098} C_VEL
LIN {X 0,Y 285.917,Z 695.485,A -85,B 0,C 180,E1 -19568.118,E2 -19568.118} C_VEL
LIN {X 0,Y 289.73,Z 676.521,A -85,B 0,C 180,E1 -19569.366,E2 -19569.366} C_VEL
LIN {X 0,Y 291.537,Z 663.086,A -85,B 0,C 180,E1 -19570.4,E2 -19570.4} C_VEL
LIN {X 0,Y 293.149,Z 649.561,A -85,B 0,C 180,E1 -19571.767,E2 -19571.767} C_VEL
LIN {X 0,Y 294.531,Z 639.17,A -85,B 0,C 180,E1 -19573.031,E2 -19573.031} C_VEL
LIN {X 0,Y 294.282,Z 637.305,A -85,B 0,C 180,E1 -19574.576,E2 -19574.576} C_VEL
LIN {X 0,Y 294.537,Z 637.337,A -85,B 0,C 180,E1 -19577.318,E2 -19577.318} C_VEL
LIN {X 0,Y 295.894,Z 641.107,A -85,B 0,C 180,E1 -19580.111,E2 -19580.111} C_VEL
LIN {X 0,Y 296.473,Z 642.62,A -85,B 0,C 180,E1 -19580.85,E2 -19580.85} C_VEL
LIN {X 0,Y 294.018,Z 658.844,A -85,B 0,C 180,E1 -19581.809,E2 -19581.809} C_VEL
LIN {X 0,Y 291.114,Z 672.699,A -85,B 0,C 180,E1 -19582.875,E2 -19582.875} C_VEL
LIN {X 0,Y 286.878,Z 687.699,A -85,B 0,C 180,E1 -19584.352,E2 -19584.352} C_VEL
LIN {X 0,Y 282.657,Z 699.976,A -85,B 0,C 180,E1 -19585.875,E2 -19585.875} C_VEL
LIN {X 0,Y 277.382,Z 712.67,A -85,B 0,C 180,E1 -19587.854,E2 -19587.854} C_VEL
LIN {X 0,Y 272.503,Z 722.785,A -85,B 0,C 180,E1 -19589.806,E2 -19589.806} C_VEL
LIN {X 0,Y 267.185,Z 732.475,A -85,B 0,C 180,E1 -19592.166,E2 -19592.166} C_VEL
LIN {X 0,Y 262.1,Z 740.472,A -85,B 0,C 180,E1 -19594.593,E2 -19594.593} C_VEL
LIN {X 0,Y 256.832,Z 747.829,A -85,B 0,C 180,E1 -19597.474,E2 -19597.474} C_VEL
LIN {X 0,Y 252.125,Z 753.532,A -85,B 0,C 180,E1 -19600.457,E2 -19600.457} C_VEL
LIN {X 0,Y 248.013,Z 757.796,A -85,B 0,C 180,E1 -19603.538,E2 -19603.538} C_VEL
LIN {X 0,Y 244.369,Z 760.73,A -85,B 0,C 180,E1 -19606.698,E2 -19606.698} C_VEL
LIN {X 0,Y 241.577,Z 762.326,A -85,B 0,C 180,E1 -19609.947,E2 -19609.947} C_VEL
LIN {X 0,Y 239.196,Z 762.751,A -85,B 0,C 180,E1 -19613.25,E2 -19613.25} C_VEL
LIN {X 0,Y 237.527,Z 761.915,A -85,B 0,C 180,E1 -19616.607,E2 -19616.607} C_VEL
LIN {X 0,Y 236.335,Z 759.869,A -85,B 0,C 180,E1 -19619.999,E2 -19619.999} C_VEL
LIN {X 0,Y 235.536,Z 756.57,A -85,B 0,C 180,E1 -19623.42,E2 -19623.42} C_VEL
LIN {X 0,Y 235.366,Z 751.922,A -85,B 0,C 180,E1 -19626.859,E2 -19626.859} C_VEL
LIN {X 0,Y 235.58,Z 745.81,A -85,B 0,C 180,E1 -19630.311,E2 -19630.311} C_VEL
LIN {X 0,Y 236.024,Z 739.081,A -85,B 0,C 180,E1 -19633.342,E2 -19633.342} C_VEL
LIN {X 0,Y 236.88,Z 730.864,A -85,B 0,C 180,E1 -19636.37,E2 -19636.37} C_VEL
LIN {X 0,Y 238.026,Z 721.042,A -85,B 0,C 180,E1 -19639.354,E2 -19639.354} C_VEL
LIN {X 0,Y 239.307,Z 710.61,A -85,B 0,C 180,E1 -19641.989,E2 -19641.989} C_VEL
LIN {X 0,Y 240.914,Z 698.532,A -85,B 0,C 180,E1 -19644.521,E2 -19644.521} C_VEL
LIN {X 0,Y 242.42,Z 686.001,A -85,B 0,C 180,E1 -19646.702,E2 -19646.702} C_VEL
LIN {X 0,Y 243.964,Z 672.661,A -85,B 0,C 180,E1 -19648.614,E2 -19648.614} C_VEL
LIN {X 0,Y 245.378,Z 657.897,A -85,B 0,C 180,E1 -19650.318,E2 -19650.318} C_VEL
LIN {X 0,Y 246.457,Z 643.888,A -85,B 0,C 180,E1 -19651.598,E2 -19651.598} C_VEL
LIN {X 0,Y 247.425,Z 627.757,A -85,B 0,C 180,E1 -19652.704,E2 -19652.704} C_VEL
LIN {X 0,Y 248.068,Z 608.588,A -85,B 0,C 180,E1 -19653.633,E2 -19653.633} C_VEL
LIN {X 0,Y 234.999,Z 571.213,A -85,B 0,C 180,E1 -19656.394,E2 -19656.394} C_VEL
LIN {X 0,Y 234.943,Z 571.217,A -85,B 0,C 180,E1 -19658.943,E2 -19658.943} C_VEL
LIN {X 0,Y 234.888,Z 571.224,A -85,B 0,C 180,E1 -19663.485,E2 -19663.485} C_VEL
LIN {X 0,Y 234.889,Z 571.225,A -85,B 0,C 180,E1 -19666.513,E2 -19666.513} C_VEL
LIN {X 0,Y 234.955,Z 571.216,A -85,B 0,C 180,E1 -19671.085,E2 -19671.085} C_VEL
LIN {X 0,Y 234.961,Z 571.214,A -85,B 0,C 180,E1 -19675.366,E2 -19675.366} C_VEL
LIN {X 0,Y 234.923,Z 571.219,A -85,B 0,C 180,E1 -19679.43,E2 -19679.43} C_VEL
LIN {X 0,Y 234.993,Z 571.211,A -85,B 0,C 180,E1 -19683.793,E2 -19683.793} C_VEL
LIN {X 0,Y 235.011,Z 571.211,A -85,B 0,C 180,E1 -19688.969,E2 -19688.969} C_VEL
LIN {X 0,Y 235.095,Z 571.199,A -85,B 0,C 180,E1 -19693.058,E2 -19693.058} C_VEL
LIN {X 0,Y 235.146,Z 571.191,A -85,B 0,C 180,E1 -19697.923,E2 -19697.923} C_VEL
LIN {X 0,Y 235.389,Z 571.162,A -85,B 0,C 180,E1 -19701.414,E2 -19701.414} C_VEL
LIN {X 0,Y 235.404,Z 571.16,A -85,B 0,C 180,E1 -19703.14,E2 -19703.14} C_VEL
LIN {X 0,Y 235.595,Z 571.136,A -85,B 0,C 180,E1 -19708.29,E2 -19708.29} C_VEL
LIN {X 0,Y 235.594,Z 571.135,A -85,B 0,C 180,E1 -19711.708,E2 -19711.708} C_VEL
LIN {X 0,Y 235.403,Z 571.161,A -85,B 0,C 180,E1 -19716.858,E2 -19716.858} C_VEL
LIN {X 0,Y 235.251,Z 571.177,A -85,B 0,C 180,E1 -19720.325,E2 -19720.325} C_VEL
LIN {X 0,Y 235.111,Z 571.199,A -85,B 0,C 180,E1 -19725.605,E2 -19725.605} C_VEL
LIN {X 0,Y 235.016,Z 571.21,A -85,B 0,C 180,E1 -19729.204,E2 -19729.204} C_VEL
LIN {X 0,Y 234.977,Z 571.212,A -85,B 0,C 180,E1 -19732.88,E2 -19732.88} C_VEL
LIN {X 0,Y 234.965,Z 571.214,A -85,B 0,C 180,E1 -19736.657,E2 -19736.657} C_VEL
LIN {X 0,Y 234.928,Z 571.217,A -85,B 0,C 180,E1 -19740.567,E2 -19740.567} C_VEL
LIN {X 0,Y 234.956,Z 571.216,A -85,B 0,C 180,E1 -19744.632,E2 -19744.632} C_VEL
LIN {X 0,Y 234.962,Z 571.215,A -85,B 0,C 180,E1 -19748.952,E2 -19748.952} C_VEL
LIN {X 0,Y 234.976,Z 571.215,A -85,B 0,C 180,E1 -19753.464,E2 -19753.464} C_VEL
LIN {X 0,Y 235.017,Z 571.212,A -85,B 0,C 180,E1 -19755.931,E2 -19755.931} C_VEL
LIN {X 0,Y 247.161,Z 604.86,A -85,B 0,C 180,E1 -19758.342,E2 -19758.342} C_VEL
LIN {X 0,Y 246.21,Z 639.045,A -85,B 0,C 180,E1 -19759.811,E2 -19759.811} C_VEL
LIN {X 0,Y 245.447,Z 653.125,A -85,B 0,C 180,E1 -19760.736,E2 -19760.736} C_VEL
LIN {X 0,Y 244.29,Z 667.807,A -85,B 0,C 180,E1 -19762.053,E2 -19762.053} C_VEL
LIN {X 0,Y 243.108,Z 680.74,A -85,B 0,C 180,E1 -19763.556,E2 -19763.556} C_VEL
LIN {X 0,Y 241.568,Z 693.641,A -85,B 0,C 180,E1 -19765.437,E2 -19765.437} C_VEL
LIN {X 0,Y 240.246,Z 705.024,A -85,B 0,C 180,E1 -19767.485,E2 -19767.485} C_VEL
LIN {X 0,Y 238.757,Z 716.389,A -85,B 0,C 180,E1 -19769.974,E2 -19769.974} C_VEL
LIN {X 0,Y 237.51,Z 726.041,A -85,B 0,C 180,E1 -19772.584,E2 -19772.584} C_VEL
LIN {X 0,Y 236.465,Z 734.612,A -85,B 0,C 180,E1 -19775.413,E2 -19775.413} C_VEL
LIN {X 0,Y 235.764,Z 741.557,A -85,B 0,C 180,E1 -19778.234,E2 -19778.234} C_VEL
LIN {X 0,Y 235.34,Z 746.698,A -85,B 0,C 180,E1 -19780.823,E2 -19780.823} C_VEL
LIN {X 0,Y 235.198,Z 750.213,A -85,B 0,C 180,E1 -19782.975,E2 -19782.975} C_VEL
LIN {X 0,Y 235.324,Z 754.253,A -85,B 0,C 180,E1 -19786.178,E2 -19786.178} C_VEL
LIN {X 0,Y 235.922,Z 757.234,A -85,B 0,C 180,E1 -19789.705,E2 -19789.705} C_VEL
LIN {X 0,Y 236.385,Z 758.161,A -85,B 0,C 180,E1 -19791.452,E2 -19791.452} C_VEL
LIN {X 0,Y 237.807,Z 758.83,A -85,B 0,C 180,E1 -19794.914,E2 -19794.914} C_VEL
LIN {X 0,Y 239.732,Z 758.064,A -85,B 0,C 180,E1 -19798.321,E2 -19798.321} C_VEL
LIN {X 0,Y 242.318,Z 755.838,A -85,B 0,C 180,E1 -19801.663,E2 -19801.663} C_VEL
LIN {X 0,Y 245.503,Z 752.027,A -85,B 0,C 180,E1 -19804.927,E2 -19804.927} C_VEL
LIN {X 0,Y 248.28,Z 748.019,A -85,B 0,C 180,E1 -19807.406,E2 -19807.406} C_VEL
LIN {X 0,Y 251.256,Z 743.273,A -85,B 0,C 180,E1 -19809.662,E2 -19809.662} C_VEL
LIN {X 0,Y 255.296,Z 736.035,A -85,B 0,C 180,E1 -19812.319,E2 -19812.319} C_VEL
LIN {X 0,Y 259.588,Z 727.145,A -85,B 0,C 180,E1 -19814.905,E2 -19814.905} C_VEL
LIN {X 0,Y 263.582,Z 717.613,A -85,B 0,C 180,E1 -19817.056,E2 -19817.056} C_VEL
LIN {X 0,Y 267.707,Z 706.356,A -85,B 0,C 180,E1 -19819.078,E2 -19819.078} C_VEL
LIN {X 0,Y 271.131,Z 695.185,A -85,B 0,C 180,E1 -19820.682,E2 -19820.682} C_VEL
LIN {X 0,Y 274.431,Z 681.825,A -85,B 0,C 180,E1 -19822.194,E2 -19822.194} C_VEL
LIN {X 0,Y 276.835,Z 668.876,A -85,B 0,C 180,E1 -19823.371,E2 -19823.371} C_VEL
LIN {X 0,Y 278.64,Z 655.16,A -85,B 0,C 180,E1 -19824.283,E2 -19824.283} C_VEL
LIN {X 0,Y 279.009,Z 651.371,A -85,B 0,C 180,E1 -19824.494,E2 -19824.494} C_VEL
LIN {X 0,Y 279.22,Z 646.18,A -85,B 0,C 180,E1 -19824.85,E2 -19824.85} C_VEL
LIN {X 0,Y 278.944,Z 641.315,A -85,B 0,C 180,E1 -19825.363,E2 -19825.363} C_VEL
LIN {X 0,Y 278.224,Z 636.997,A -85,B 0,C 180,E1 -19826.026,E2 -19826.026} C_VEL
LIN {X 0,Y 277.091,Z 633.483,A -85,B 0,C 180,E1 -19826.844,E2 -19826.844} C_VEL
LIN {X 0,Y 274.741,Z 628.635,A -85,B 0,C 180,E1 -19828.516,E2 -19828.516} C_VEL
LIN {X 0,Y 272.849,Z 625.079,A -85,B 0,C 180,E1 -19830.094,E2 -19830.094} C_VEL
LIN {X 0,Y 271.822,Z 623.124,A -85,B 0,C 180,E1 -19831.139,E2 -19831.139} C_VEL
LIN {X 0,Y 270.04,Z 619.711,A -85,B 0,C 180,E1 -19833.439,E2 -19833.439} C_VEL
LIN {X 0,Y 268.592,Z 618.099,A -85,B 0,C 180,E1 -19836.472,E2 -19836.472} C_VEL
LIN {X 0,Y 268.341,Z 617.855,A -85,B 0,C 180,E1 -19838.946,E2 -19838.946} C_VEL
LIN {X 0,Y 269.189,Z 619.037,A -85,B 0,C 180,E1 -19841.956,E2 -19841.956} C_VEL
LIN {X 0,Y 269.888,Z 619.84,A -85,B 0,C 180,E1 -19843.188,E2 -19843.188} C_VEL
LIN {X 0,Y 270.566,Z 621.854,A -85,B 0,C 180,E1 -19844.337,E2 -19844.337} C_VEL
LIN {X 0,Y 271.166,Z 628.323,A -85,B 0,C 180,E1 -19846.007,E2 -19846.007} C_VEL
LIN {X 0,Y 271.536,Z 633.946,A -85,B 0,C 180,E1 -19847.129,E2 -19847.129} C_VEL
LIN {X 0,Y 271.244,Z 648.478,A -85,B 0,C 180,E1 -19848.865,E2 -19848.865} C_VEL
LIN {X 0,Y 270.936,Z 664.691,A -85,B 0,C 180,E1 -19850.522,E2 -19850.522} C_VEL
LIN {X 0,Y 270.537,Z 673.971,A -85,B 0,C 180,E1 -19851.297,E2 -19851.297} C_VEL
LIN {X 0,Y 268.946,Z 697.983,A -85,B 0,C 180,E1 -19853.058,E2 -19853.058} C_VEL
LIN {X 0,Y 265.983,Z 712.813,A -85,B 0,C 180,E1 -19853.888,E2 -19853.888} C_VEL
LIN {X 0,Y 261.792,Z 728.097,A -85,B 0,C 180,E1 -19854.984,E2 -19854.984} C_VEL
LIN {X 0,Y 257.019,Z 742.619,A -85,B 0,C 180,E1 -19856.378,E2 -19856.378} C_VEL
LIN {X 0,Y 252.08,Z 755.722,A -85,B 0,C 180,E1 -19858.015,E2 -19858.015} C_VEL
LIN {X 0,Y 247.576,Z 766.574,A -85,B 0,C 180,E1 -19859.745,E2 -19859.745} C_VEL
LIN {X 0,Y 242.728,Z 777.511,A -85,B 0,C 180,E1 -19861.934,E2 -19861.934} C_VEL
LIN {X 0,Y 238.48,Z 786.629,A -85,B 0,C 180,E1 -19864.236,E2 -19864.236} C_VEL
LIN {X 0,Y 234.938,Z 794.339,A -85,B 0,C 180,E1 -19866.65,E2 -19866.65} C_VEL
LIN {X 0,Y 231.579,Z 801.764,A -85,B 0,C 180,E1 -19869.575,E2 -19869.575} C_VEL
LIN {X 0,Y 229.401,Z 806.952,A -85,B 0,C 180,E1 -19872.161,E2 -19872.161} C_VEL
LIN {X 0,Y 227.939,Z 811.14,A -85,B 0,C 180,E1 -19874.808,E2 -19874.808} C_VEL
LIN {X 0,Y 226.994,Z 814.42,A -85,B 0,C 180,E1 -19877.484,E2 -19877.484} C_VEL
LIN {X 0,Y 226.768,Z 817.442,A -85,B 0,C 180,E1 -19881.087,E2 -19881.087} C_VEL
LIN {X 0,Y 226.945,Z 818.371,A -85,B 0,C 180,E1 -19882.885,E2 -19882.885} C_VEL
LIN {X 0,Y 227.372,Z 818.891,A -85,B 0,C 180,E1 -19884.68,E2 -19884.68} C_VEL
LIN {X 0,Y 227.84,Z 818.966,A -85,B 0,C 180,E1 -19886.464,E2 -19886.464} C_VEL
LIN {X 0,Y 228.908,Z 818.091,A -85,B 0,C 180,E1 -19889.561,E2 -19889.561} C_VEL
LIN {X 0,Y 229.049,Z 818.092,A -85,B 0,C 180,E1 -19890.001,E2 -19890.001} C_VEL
LIN {X 0,Y 228.371,Z 819.091,A -85,B 0,C 180,E1 -19891.765,E2 -19891.765} C_VEL
LIN {X 0,Y 227.831,Z 819.67,A -85,B 0,C 180,E1 -19893.538,E2 -19893.538} C_VEL
LIN {X 0,Y 227.287,Z 819.813,A -85,B 0,C 180,E1 -19895.324,E2 -19895.324} C_VEL
LIN {X 0,Y 226.838,Z 819.476,A -85,B 0,C 180,E1 -19897.497,E2 -19897.497} C_VEL
LIN {X 0,Y 226.642,Z 817.901,A -85,B 0,C 180,E1 -19900.724,E2 -19900.724} C_VEL
LIN {X 0,Y 227.497,Z 814.791,A -85,B 0,C 180,E1 -19904.309,E2 -19904.309} C_VEL
LIN {X 0,Y 229.261,Z 810.195,A -85,B 0,C 180,E1 -19907.852,E2 -19907.852} C_VEL
LIN {X 0,Y 232.472,Z 804.103,A -85,B 0,C 180,E1 -19911.272,E2 -19911.272} C_VEL
LIN {X 0,Y 236.237,Z 797.44,A -85,B 0,C 180,E1 -19914.147,E2 -19914.147} C_VEL
LIN {X 0,Y 240.856,Z 789.393,A -85,B 0,C 180,E1 -19916.891,E2 -19916.891} C_VEL
LIN {X 0,Y 246.289,Z 779.821,A -85,B 0,C 180,E1 -19919.489,E2 -19919.489} C_VEL
LIN {X 0,Y 251.59,Z 770.203,A -85,B 0,C 180,E1 -19921.586,E2 -19921.586} C_VEL
LIN {X 0,Y 258.68,Z 756.918,A -85,B 0,C 180,E1 -19923.847,E2 -19923.847} C_VEL
LIN {X 0,Y 265.363,Z 743.252,A -85,B 0,C 180,E1 -19925.639,E2 -19925.639} C_VEL
LIN {X 0,Y 271.311,Z 729.827,A -85,B 0,C 180,E1 -19927.033,E2 -19927.033} C_VEL
LIN {X 0,Y 277.185,Z 715.053,A -85,B 0,C 180,E1 -19928.215,E2 -19928.215} C_VEL
LIN {X 0,Y 282.823,Z 697.973,A -85,B 0,C 180,E1 -19929.322,E2 -19929.322} C_VEL
LIN {X 0,Y 287.337,Z 679.11,A -85,B 0,C 180,E1 -19930.598,E2 -19930.598} C_VEL
LIN {X 0,Y 289.67,Z 665.454,A -85,B 0,C 180,E1 -19931.675,E2 -19931.675} C_VEL
LIN {X 0,Y 291.609,Z 652.434,A -85,B 0,C 180,E1 -19933,E2 -19933} C_VEL
LIN {X 0,Y 292.788,Z 645.122,A -85,B 0,C 180,E1 -19933.895,E2 -19933.895} C_VEL
LIN {X 0,Y 292.771,Z 644.212,A -85,B 0,C 180,E1 -19934.585,E2 -19934.585} C_VEL
LIN {X 0,Y 293.016,Z 644.432,A -85,B 0,C 180,E1 -19937.328,E2 -19937.328} C_VEL
LIN {X 0,Y 294.072,Z 647.729,A -85,B 0,C 180,E1 -19939.741,E2 -19939.741} C_VEL
LIN {X 0,Y 291.441,Z 662.825,A -85,B 0,C 180,E1 -19940.685,E2 -19940.685} C_VEL
LIN {X 0,Y 288.196,Z 676.284,A -85,B 0,C 180,E1 -19941.771,E2 -19941.771} C_VEL
LIN {X 0,Y 284.037,Z 689.962,A -85,B 0,C 180,E1 -19943.128,E2 -19943.128} C_VEL
LIN {X 0,Y 279.437,Z 702.108,A -85,B 0,C 180,E1 -19944.657,E2 -19944.657} C_VEL
LIN {X 0,Y 275.005,Z 712.334,A -85,B 0,C 180,E1 -19946.231,E2 -19946.231} C_VEL
LIN {X 0,Y 269.737,Z 722.605,A -85,B 0,C 180,E1 -19948.155,E2 -19948.155} C_VEL
LIN {X 0,Y 264.782,Z 731.313,A -85,B 0,C 180,E1 -19950.153,E2 -19950.153} C_VEL
LIN {X 0,Y 259.29,Z 739.69,A -85,B 0,C 180,E1 -19952.562,E2 -19952.562} C_VEL
LIN {X 0,Y 254.908,Z 745.719,A -85,B 0,C 180,E1 -19954.7,E2 -19954.7} C_VEL
LIN {X 0,Y 249.51,Z 752.178,A -85,B 0,C 180,E1 -19957.65,E2 -19957.65} C_VEL
LIN {X 0,Y 244.698,Z 757.188,A -85,B 0,C 180,E1 -19960.713,E2 -19960.713} C_VEL
LIN {X 0,Y 241.539,Z 759.949,A -85,B 0,C 180,E1 -19963.083,E2 -19963.083} C_VEL
LIN {X 0,Y 237.709,Z 762.582,A -85,B 0,C 180,E1 -19966.318,E2 -19966.318} C_VEL
LIN {X 0,Y 234.784,Z 763.883,A -85,B 0,C 180,E1 -19969.653,E2 -19969.653} C_VEL
LIN {X 0,Y 232.272,Z 764.022,A -85,B 0,C 180,E1 -19973.048,E2 -19973.048} C_VEL
LIN {X 0,Y 230.533,Z 762.918,A -85,B 0,C 180,E1 -19976.504,E2 -19976.504} C_VEL
LIN {X 0,Y 229.271,Z 760.6,A -85,B 0,C 180,E1 -19979.999,E2 -19979.999} C_VEL
LIN {X 0,Y 228.441,Z 757.023,A -85,B 0,C 180,E1 -19983.527,E2 -19983.527} C_VEL
LIN {X 0,Y 228.292,Z 751.884,A -85,B 0,C 180,E1 -19987.183,E2 -19987.183} C_VEL
LIN {X 0,Y 228.515,Z 745.619,A -85,B 0,C 180,E1 -19990.633,E2 -19990.633} C_VEL
LIN {X 0,Y 229.01,Z 738.586,A -85,B 0,C 180,E1 -19993.758,E2 -19993.758} C_VEL
LIN {X 0,Y 229.972,Z 730.054,A -85,B 0,C 180,E1 -19996.876,E2 -19996.876} C_VEL
LIN {X 0,Y 231.191,Z 719.67,A -85,B 0,C 180,E1 -19999.997,E2 -19999.997} C_VEL
LIN {X 0,Y 232.532,Z 708.923,A -85,B 0,C 180,E1 -20002.665,E2 -20002.665} C_VEL
LIN {X 0,Y 234.191,Z 696.565,A -85,B 0,C 180,E1 -20005.198,E2 -20005.198} C_VEL
LIN {X 0,Y 235.83,Z 682.869,A -85,B 0,C 180,E1 -20007.51,E2 -20007.51} C_VEL
LIN {X 0,Y 237.256,Z 670.254,A -85,B 0,C 180,E1 -20009.258,E2 -20009.258} C_VEL
LIN {X 0,Y 238.697,Z 655.244,A -85,B 0,C 180,E1 -20010.945,E2 -20010.945} C_VEL
LIN {X 0,Y 239.793,Z 640.859,A -85,B 0,C 180,E1 -20012.211,E2 -20012.211} C_VEL
LIN {X 0,Y 240.67,Z 625.284,A -85,B 0,C 180,E1 -20013.234,E2 -20013.234} C_VEL
LIN {X 0,Y 241.11,Z 609.845,A -85,B 0,C 180,E1 -20013.995,E2 -20013.995} C_VEL
LIN {X 0,Y 227.935,Z 572.09,A -85,B 0,C 180,E1 -20016.876,E2 -20016.876} C_VEL
LIN {X 0,Y 227.827,Z 572.105,A -85,B 0,C 180,E1 -20020.375,E2 -20020.375} C_VEL
LIN {X 0,Y 227.834,Z 572.103,A -85,B 0,C 180,E1 -20025.191,E2 -20025.191} C_VEL
LIN {X 0,Y 227.835,Z 572.1,A -85,B 0,C 180,E1 -20029.624,E2 -20029.624} C_VEL
LIN {X 0,Y 227.9,Z 572.096,A -85,B 0,C 180,E1 -20034.131,E2 -20034.131} C_VEL
LIN {X 0,Y 227.869,Z 572.098,A -85,B 0,C 180,E1 -20038.376,E2 -20038.376} C_VEL
LIN {X 0,Y 227.879,Z 572.1,A -85,B 0,C 180,E1 -20042.443,E2 -20042.443} C_VEL
LIN {X 0,Y 227.913,Z 572.092,A -85,B 0,C 180,E1 -20046.366,E2 -20046.366} C_VEL
LIN {X 0,Y 227.942,Z 572.09,A -85,B 0,C 180,E1 -20050.173,E2 -20050.173} C_VEL
LIN {X 0,Y 228.057,Z 572.073,A -85,B 0,C 180,E1 -20053.897,E2 -20053.897} C_VEL
LIN {X 0,Y 228.17,Z 572.062,A -85,B 0,C 180,E1 -20059.349,E2 -20059.349} C_VEL
LIN {X 0,Y 228.357,Z 572.039,A -85,B 0,C 180,E1 -20062.928,E2 -20062.928} C_VEL
LIN {X 0,Y 228.553,Z 572.013,A -85,B 0,C 180,E1 -20068.237,E2 -20068.237} C_VEL
LIN {X 0,Y 228.553,Z 572.012,A -85,B 0,C 180,E1 -20071.761,E2 -20071.761} C_VEL
LIN {X 0,Y 228.355,Z 572.04,A -85,B 0,C 180,E1 -20077.07,E2 -20077.07} C_VEL
LIN {X 0,Y 228.169,Z 572.06,A -85,B 0,C 180,E1 -20080.649,E2 -20080.649} C_VEL
LIN {X 0,Y 228.055,Z 572.076,A -85,B 0,C 180,E1 -20086.101,E2 -20086.101} C_VEL
LIN {X 0,Y 227.951,Z 572.087,A -85,B 0,C 180,E1 -20089.824,E2 -20089.824} C_VEL
LIN {X 0,Y 227.92,Z 572.095,A -85,B 0,C 180,E1 -20093.631,E2 -20093.631} C_VEL
LIN {X 0,Y 227.881,Z 572.1,A -85,B 0,C 180,E1 -20097.554,E2 -20097.554} C_VEL
LIN {X 0,Y 227.869,Z 572.1,A -85,B 0,C 180,E1 -20101.621,E2 -20101.621} C_VEL
LIN {X 0,Y 227.897,Z 572.099,A -85,B 0,C 180,E1 -20105.867,E2 -20105.867} C_VEL
LIN {X 0,Y 227.876,Z 572.099,A -85,B 0,C 180,E1 -20110.364,E2 -20110.364} C_VEL
LIN {X 0,Y 227.912,Z 572.094,A -85,B 0,C 180,E1 -20114.828,E2 -20114.828} C_VEL
LIN {X 0,Y 227.927,Z 572.092,A -85,B 0,C 180,E1 -20115.403,E2 -20115.403} C_VEL
LIN {X 0,Y 240.22,Z 606.031,A -85,B 0,C 180,E1 -20117.923,E2 -20117.923} C_VEL
LIN {X 0,Y 239.284,Z 640.037,A -85,B 0,C 180,E1 -20119.446,E2 -20119.446} C_VEL
LIN {X 0,Y 238.515,Z 654.376,A -85,B 0,C 180,E1 -20120.418,E2 -20120.418} C_VEL
LIN {X 0,Y 237.276,Z 669.376,A -85,B 0,C 180,E1 -20121.808,E2 -20121.808} C_VEL
LIN {X 0,Y 235.971,Z 682.846,A -85,B 0,C 180,E1 -20123.441,E2 -20123.441} C_VEL
LIN {X 0,Y 234.492,Z 695.041,A -85,B 0,C 180,E1 -20125.289,E2 -20125.289} C_VEL
LIN {X 0,Y 233.137,Z 706.368,A -85,B 0,C 180,E1 -20127.392,E2 -20127.392} C_VEL
LIN {X 0,Y 231.637,Z 717.71,A -85,B 0,C 180,E1 -20129.96,E2 -20129.96} C_VEL
LIN {X 0,Y 230.318,Z 727.672,A -85,B 0,C 180,E1 -20132.761,E2 -20132.761} C_VEL
LIN {X 0,Y 229.318,Z 735.828,A -85,B 0,C 180,E1 -20135.561,E2 -20135.561} C_VEL
LIN {X 0,Y 228.661,Z 742.501,A -85,B 0,C 180,E1 -20138.358,E2 -20138.358} C_VEL
LIN {X 0,Y 228.228,Z 747.893,A -85,B 0,C 180,E1 -20141.136,E2 -20141.136} C_VEL
LIN {X 0,Y 228.125,Z 752.175,A -85,B 0,C 180,E1 -20143.904,E2 -20143.904} C_VEL
LIN {X 0,Y 228.238,Z 754.493,A -85,B 0,C 180,E1 -20145.74,E2 -20145.74} C_VEL
LIN {X 0,Y 228.418,Z 756.385,A -85,B 0,C 180,E1 -20147.563,E2 -20147.563} C_VEL
LIN {X 0,Y 229.265,Z 758.94,A -85,B 0,C 180,E1 -20151.184,E2 -20151.184} C_VEL
LIN {X 0,Y 230.694,Z 760.03,A -85,B 0,C 180,E1 -20154.757,E2 -20154.757} C_VEL
LIN {X 0,Y 232.671,Z 759.669,A -85,B 0,C 180,E1 -20158.27,E2 -20158.27} C_VEL
LIN {X 0,Y 235.337,Z 757.789,A -85,B 0,C 180,E1 -20161.712,E2 -20161.712} C_VEL
LIN {X 0,Y 238.617,Z 754.441,A -85,B 0,C 180,E1 -20165.07,E2 -20165.07} C_VEL
LIN {X 0,Y 241.791,Z 750.37,A -85,B 0,C 180,E1 -20167.835,E2 -20167.835} C_VEL
LIN {X 0,Y 245.766,Z 744.634,A -85,B 0,C 180,E1 -20170.713,E2 -20170.713} C_VEL
LIN {X 0,Y 250.034,Z 737.483,A -85,B 0,C 180,E1 -20173.409,E2 -20173.409} C_VEL
LIN {X 0,Y 254.641,Z 728.58,A -85,B 0,C 180,E1 -20176.022,E2 -20176.022} C_VEL
LIN {X 0,Y 258.888,Z 719.244,A -85,B 0,C 180,E1 -20178.173,E2 -20178.173} C_VEL
LIN {X 0,Y 263.411,Z 707.548,A -85,B 0,C 180,E1 -20180.295,E2 -20180.295} C_VEL
LIN {X 0,Y 266.513,Z 698.222,A -85,B 0,C 180,E1 -20181.666,E2 -20181.666} C_VEL
LIN {X 0,Y 269.615,Z 687.039,A -85,B 0,C 180,E1 -20183.018,E2 -20183.018} C_VEL
LIN {X 0,Y 272.635,Z 672.995,A -85,B 0,C 180,E1 -20184.359,E2 -20184.359} C_VEL
LIN {X 0,Y 274.667,Z 659.959,A -85,B 0,C 180,E1 -20185.33,E2 -20185.33} C_VEL
LIN {X 0,Y 277.156,Z 636.226,A -85,B 0,C 180,E1 -20186.547,E2 -20186.547} C_VEL
LIN {X 0,Y 277.346,Z 634.033,A -85,B 0,C 180,E1 -20186.675,E2 -20186.675} C_VEL
LIN {X 0,Y 277.091,Z 633.483,A -85,B 0,C 180,E1 -20186.844,E2 -20186.844} C_VEL
LIN {X 0,Y 276.021,Z 631.713,A -85,B 0,C 180,E1 -20187.536,E2 -20187.536} C_VEL
LIN {X 0,Y 274.191,Z 630.248,A -85,B 0,C 180,E1 -20188.671,E2 -20188.671} C_VEL
LIN {X 0,Y 270.144,Z 629.134,A -85,B 0,C 180,E1 -20191.515,E2 -20191.515} C_VEL
LIN {X 0,Y 268.952,Z 628.058,A -85,B 0,C 180,E1 -20192.756,E2 -20192.756} C_VEL
LIN {X 0,Y 268.68,Z 627.437,A -85,B 0,C 180,E1 -20193.161,E2 -20193.161} C_VEL
LIN {X 0,Y 268.286,Z 626.357,A -85,B 0,C 180,E1 -20193.856,E2 -20193.856} C_VEL
LIN {X 0,Y 266.94,Z 624.869,A -85,B 0,C 180,E1 -20197.269,E2 -20197.269} C_VEL
LIN {X 0,Y 267.018,Z 625.077,A -85,B 0,C 180,E1 -20199.94,E2 -20199.94} C_VEL
LIN {X 0,Y 268.227,Z 626.692,A -85,B 0,C 180,E1 -20202.942,E2 -20202.942} C_VEL
LIN {X 0,Y 268.586,Z 628.28,A -85,B 0,C 180,E1 -20203.733,E2 -20203.733} C_VEL
LIN {X 0,Y 268.856,Z 633.385,A -85,B 0,C 180,E1 -20205.079,E2 -20205.079} C_VEL
LIN {X 0,Y 269.039,Z 637.86,A -85,B 0,C 180,E1 -20205.98,E2 -20205.98} C_VEL
LIN {X 0,Y 268.407,Z 652.345,A -85,B 0,C 180,E1 -20207.731,E2 -20207.731} C_VEL
LIN {X 0,Y 267.749,Z 667.705,A -85,B 0,C 180,E1 -20209.324,E2 -20209.324} C_VEL
LIN {X 0,Y 267.3,Z 675.656,A -85,B 0,C 180,E1 -20210,E2 -20210} C_VEL
LIN {X 0,Y 265.238,Z 699.176,A -85,B 0,C 180,E1 -20211.784,E2 -20211.784} C_VEL
LIN {X 0,Y 261.701,Z 714.573,A -85,B 0,C 180,E1 -20212.706,E2 -20212.706} C_VEL
LIN {X 0,Y 257.291,Z 729.115,A -85,B 0,C 180,E1 -20213.795,E2 -20213.795} C_VEL
LIN {X 0,Y 252.319,Z 743.052,A -85,B 0,C 180,E1 -20215.181,E2 -20215.181} C_VEL
LIN {X 0,Y 247.169,Z 755.679,A -85,B 0,C 180,E1 -20216.816,E2 -20216.816} C_VEL
LIN {X 0,Y 241.58,Z 768.162,A -85,B 0,C 180,E1 -20218.912,E2 -20218.912} C_VEL
LIN {X 0,Y 236.553,Z 778.53,A -85,B 0,C 180,E1 -20221.134,E2 -20221.134} C_VEL
LIN {X 0,Y 232.132,Z 787.246,A -85,B 0,C 180,E1 -20223.477,E2 -20223.477} C_VEL
LIN {X 0,Y 227.872,Z 795.637,A -85,B 0,C 180,E1 -20226.364,E2 -20226.364} C_VEL
LIN {X 0,Y 224.926,Z 801.626,A -85,B 0,C 180,E1 -20228.942,E2 -20228.942} C_VEL
LIN {X 0,Y 222.6,Z 806.566,A -85,B 0,C 180,E1 -20231.597,E2 -20231.597} C_VEL
LIN {X 0,Y 220.629,Z 811.688,A -85,B 0,C 180,E1 -20235.237,E2 -20235.237} C_VEL
LIN {X 0,Y 219.712,Z 815.258,A -85,B 0,C 180,E1 -20238.936,E2 -20238.936} C_VEL
LIN {X 0,Y 219.891,Z 817.258,A -85,B 0,C 180,E1 -20242.656,E2 -20242.656} C_VEL
LIN {X 0,Y 220.306,Z 817.677,A -85,B 0,C 180,E1 -20244.509,E2 -20244.509} C_VEL
LIN {X 0,Y 220.819,Z 817.677,A -85,B 0,C 180,E1 -20246.352,E2 -20246.352} C_VEL
LIN {X 0,Y 222.036,Z 816.544,A -85,B 0,C 180,E1 -20249.774,E2 -20249.774} C_VEL
LIN {X 0,Y 222.126,Z 816.435,A -85,B 0,C 180,E1 -20250.001,E2 -20250.001} C_VEL
LIN {X 0,Y 221.432,Z 817.553,A -85,B 0,C 180,E1 -20251.82,E2 -20251.82} C_VEL
LIN {X 0,Y 220.831,Z 818.216,A -85,B 0,C 180,E1 -20253.65,E2 -20253.65} C_VEL
LIN {X 0,Y 219.858,Z 818.301,A -85,B 0,C 180,E1 -20257.347,E2 -20257.347} C_VEL
LIN {X 0,Y 219.629,Z 816.875,A -85,B 0,C 180,E1 -20261.07,E2 -20261.07} C_VEL
LIN {X 0,Y 220.548,Z 814.027,A -85,B 0,C 180,E1 -20264.77,E2 -20264.77} C_VEL
LIN {X 0,Y 222.614,Z 809.358,A -85,B 0,C 180,E1 -20268.715,E2 -20268.715} C_VEL
LIN {X 0,Y 225.849,Z 804.071,A -85,B 0,C 180,E1 -20271.928,E2 -20271.928} C_VEL
LIN {X 0,Y 230.419,Z 796.816,A -85,B 0,C 180,E1 -20275.279,E2 -20275.279} C_VEL
LIN {X 0,Y 236.061,Z 787.805,A -85,B 0,C 180,E1 -20278.448,E2 -20278.448} C_VEL
LIN {X 0,Y 242.847,Z 776.882,A -85,B 0,C 180,E1 -20281.395,E2 -20281.395} C_VEL
LIN {X 0,Y 248.707,Z 767.143,A -85,B 0,C 180,E1 -20283.439,E2 -20283.439} C_VEL
LIN {X 0,Y 255.724,Z 754.799,A -85,B 0,C 180,E1 -20285.492,E2 -20285.492} C_VEL
LIN {X 0,Y 262.779,Z 741.291,A -85,B 0,C 180,E1 -20287.237,E2 -20287.237} C_VEL
LIN {X 0,Y 269.105,Z 727.976,A -85,B 0,C 180,E1 -20288.575,E2 -20288.575} C_VEL
LIN {X 0,Y 275.113,Z 713.77,A -85,B 0,C 180,E1 -20289.692,E2 -20289.692} C_VEL
LIN {X 0,Y 280.405,Z 698.976,A -85,B 0,C 180,E1 -20290.668,E2 -20290.668} C_VEL
LIN {X 0,Y 285.897,Z 678.873,A -85,B 0,C 180,E1 -20292.065,E2 -20292.065} C_VEL
LIN {X 0,Y 288.313,Z 666.996,A -85,B 0,C 180,E1 -20293.043,E2 -20293.043} C_VEL
LIN {X 0,Y 290.53,Z 654.704,A -85,B 0,C 180,E1 -20294.33,E2 -20294.33} C_VEL
LIN {X 0,Y 291.225,Z 651.149,A -85,B 0,C 180,E1 -20294.774,E2 -20294.774} C_VEL
LIN {X 0,Y 291.449,Z 651.365,A -85,B 0,C 180,E1 -20297.165,E2 -20297.165} C_VEL
LIN {X 0,Y 291.909,Z 653.286,A -85,B 0,C 180,E1 -20298.646,E2 -20298.646} C_VEL
LIN {X 0,Y 288.863,Z 667.974,A -85,B 0,C 180,E1 -20299.628,E2 -20299.628} C_VEL
LIN {X 0,Y 285.495,Z 680.292,A -85,B 0,C 180,E1 -20300.662,E2 -20300.662} C_VEL
LIN {X 0,Y 281.003,Z 693.451,A -85,B 0,C 180,E1 -20302.007,E2 -20302.007} C_VEL
LIN {X 0,Y 275.28,Z 707.232,A -85,B 0,C 180,E1 -20303.815,E2 -20303.815} C_VEL
LIN {X 0,Y 270.097,Z 717.648,A -85,B 0,C 180,E1 -20305.532,E2 -20305.532} C_VEL
LIN {X 0,Y 264.656,Z 727.343,A -85,B 0,C 180,E1 -20307.469,E2 -20307.469} C_VEL
LIN {X 0,Y 258.593,Z 736.616,A -85,B 0,C 180,E1 -20309.814,E2 -20309.814} C_VEL
LIN {X 0,Y 253.707,Z 743.332,A -85,B 0,C 180,E1 -20311.905,E2 -20311.905} C_VEL
LIN {X 0,Y 247.629,Z 750.583,A -85,B 0,C 180,E1 -20314.803,E2 -20314.803} C_VEL
LIN {X 0,Y 242.149,Z 756.274,A -85,B 0,C 180,E1 -20317.832,E2 -20317.832} C_VEL
LIN {X 0,Y 237.24,Z 760.519,A -85,B 0,C 180,E1 -20320.981,E2 -20320.981} C_VEL
LIN {X 0,Y 232.988,Z 763.437,A -85,B 0,C 180,E1 -20324.247,E2 -20324.247} C_VEL
LIN {X 0,Y 229.358,Z 765.088,A -85,B 0,C 180,E1 -20327.613,E2 -20327.613} C_VEL
LIN {X 0,Y 226.59,Z 765.502,A -85,B 0,C 180,E1 -20331.078,E2 -20331.078} C_VEL
LIN {X 0,Y 224.378,Z 764.718,A -85,B 0,C 180,E1 -20334.607,E2 -20334.607} C_VEL
LIN {X 0,Y 222.747,Z 762.733,A -85,B 0,C 180,E1 -20338.191,E2 -20338.191} C_VEL
LIN {X 0,Y 221.75,Z 759.5,A -85,B 0,C 180,E1 -20341.815,E2 -20341.815} C_VEL
LIN {X 0,Y 221.167,Z 754.962,A -85,B 0,C 180,E1 -20345.47,E2 -20345.47} C_VEL
LIN {X 0,Y 221.34,Z 748.984,A -85,B 0,C 180,E1 -20349.134,E2 -20349.134} C_VEL
LIN {X 0,Y 221.679,Z 742.394,A -85,B 0,C 180,E1 -20352.356,E2 -20352.356} C_VEL
LIN {X 0,Y 222.361,Z 734.373,A -85,B 0,C 180,E1 -20355.583,E2 -20355.583} C_VEL
LIN {X 0,Y 223.498,Z 725.08,A -85,B 0,C 180,E1 -20358.674,E2 -20358.674} C_VEL
LIN {X 0,Y 224.791,Z 714.664,A -85,B 0,C 180,E1 -20361.552,E2 -20361.552} C_VEL
LIN {X 0,Y 226.414,Z 702.729,A -85,B 0,C 180,E1 -20364.285,E2 -20364.285} C_VEL
LIN {X 0,Y 227.937,Z 690.579,A -85,B 0,C 180,E1 -20366.597,E2 -20366.597} C_VEL
LIN {X 0,Y 229.641,Z 676.335,A -85,B 0,C 180,E1 -20368.816,E2 -20368.816} C_VEL
LIN {X 0,Y 231.146,Z 662.011,A -85,B 0,C 180,E1 -20370.615,E2 -20370.615} C_VEL
LIN {X 0,Y 232.437,Z 647.088,A -85,B 0,C 180,E1 -20372.087,E2 -20372.087} C_VEL
LIN {X 0,Y 233.477,Z 630.88,A -85,B 0,C 180,E1 -20373.294,E2 -20373.294} C_VEL
LIN {X 0,Y 234.253,Z 611.467,A -85,B 0,C 180,E1 -20374.319,E2 -20374.319} C_VEL
LIN {X 0,Y 220.852,Z 572.972,A -85,B 0,C 180,E1 -20377.349,E2 -20377.349} C_VEL
LIN {X 0,Y 220.771,Z 572.983,A -85,B 0,C 180,E1 -20381.951,E2 -20381.951} C_VEL
LIN {X 0,Y 220.775,Z 572.982,A -85,B 0,C 180,E1 -20385.545,E2 -20385.545} C_VEL
LIN {X 0,Y 220.81,Z 572.979,A -85,B 0,C 180,E1 -20390.463,E2 -20390.463} C_VEL
LIN {X 0,Y 220.832,Z 572.977,A -85,B 0,C 180,E1 -20392.793,E2 -20392.793} C_VEL
LIN {X 0,Y 220.823,Z 572.973,A -85,B 0,C 180,E1 -20397.244,E2 -20397.244} C_VEL
LIN {X 0,Y 220.827,Z 572.976,A -85,B 0,C 180,E1 -20401.484,E2 -20401.484} C_VEL
LIN {X 0,Y 220.867,Z 572.968,A -85,B 0,C 180,E1 -20405.564,E2 -20405.564} C_VEL
LIN {X 0,Y 220.892,Z 572.968,A -85,B 0,C 180,E1 -20409.513,E2 -20409.513} C_VEL
LIN {X 0,Y 221.016,Z 572.951,A -85,B 0,C 180,E1 -20413.369,E2 -20413.369} C_VEL
LIN {X 0,Y 221.116,Z 572.944,A -85,B 0,C 180,E1 -20419.005,E2 -20419.005} C_VEL
LIN {X 0,Y 221.31,Z 572.917,A -85,B 0,C 180,E1 -20422.701,E2 -20422.701} C_VEL
LIN {X 0,Y 221.511,Z 572.89,A -85,B 0,C 180,E1 -20428.181,E2 -20428.181} C_VEL
LIN {X 0,Y 221.511,Z 572.888,A -85,B 0,C 180,E1 -20431.817,E2 -20431.817} C_VEL
LIN {X 0,Y 221.308,Z 572.92,A -85,B 0,C 180,E1 -20437.297,E2 -20437.297} C_VEL
LIN {X 0,Y 221.114,Z 572.94,A -85,B 0,C 180,E1 -20440.993,E2 -20440.993} C_VEL
LIN {X 0,Y 221.014,Z 572.953,A -85,B 0,C 180,E1 -20446.629,E2 -20446.629} C_VEL
LIN {X 0,Y 220.906,Z 572.962,A -85,B 0,C 180,E1 -20450.484,E2 -20450.484} C_VEL
LIN {X 0,Y 220.869,Z 572.97,A -85,B 0,C 180,E1 -20454.434,E2 -20454.434} C_VEL
LIN {X 0,Y 220.832,Z 572.973,A -85,B 0,C 180,E1 -20458.513,E2 -20458.513} C_VEL
LIN {X 0,Y 220.82,Z 572.976,A -85,B 0,C 180,E1 -20462.754,E2 -20462.754} C_VEL
LIN {X 0,Y 220.833,Z 572.976,A -85,B 0,C 180,E1 -20467.287,E2 -20467.287} C_VEL
LIN {X 0,Y 220.846,Z 572.977,A -85,B 0,C 180,E1 -20471.933,E2 -20471.933} C_VEL
LIN {X 0,Y 220.885,Z 572.969,A -85,B 0,C 180,E1 -20474.864,E2 -20474.864} C_VEL
LIN {X 0,Y 233.395,Z 607.595,A -85,B 0,C 180,E1 -20477.519,E2 -20477.519} C_VEL
LIN {X 0,Y 232.401,Z 641.207,A -85,B 0,C 180,E1 -20479.071,E2 -20479.071} C_VEL
LIN {X 0,Y 231.567,Z 655.387,A -85,B 0,C 180,E1 -20480.058,E2 -20480.058} C_VEL
LIN {X 0,Y 230.359,Z 669.761,A -85,B 0,C 180,E1 -20481.427,E2 -20481.427} C_VEL
LIN {X 0,Y 229.105,Z 682.614,A -85,B 0,C 180,E1 -20483.006,E2 -20483.006} C_VEL
LIN {X 0,Y 227.575,Z 694.919,A -85,B 0,C 180,E1 -20484.889,E2 -20484.889} C_VEL
LIN {X 0,Y 226.193,Z 706.256,A -85,B 0,C 180,E1 -20487.023,E2 -20487.023} C_VEL
LIN {X 0,Y 224.752,Z 716.954,A -85,B 0,C 180,E1 -20489.461,E2 -20489.461} C_VEL
LIN {X 0,Y 223.59,Z 725.739,A -85,B 0,C 180,E1 -20491.87,E2 -20491.87} C_VEL
LIN {X 0,Y 222.482,Z 734.494,A -85,B 0,C 180,E1 -20494.758,E2 -20494.758} C_VEL
LIN {X 0,Y 221.614,Z 742.653,A -85,B 0,C 180,E1 -20498.123,E2 -20498.123} C_VEL
LIN {X 0,Y 221.114,Z 749.09,A -85,B 0,C 180,E1 -20501.468,E2 -20501.468} C_VEL
LIN {X 0,Y 221.081,Z 753.366,A -85,B 0,C 180,E1 -20504.324,E2 -20504.324} C_VEL
LIN {X 0,Y 221.316,Z 756.652,A -85,B 0,C 180,E1 -20507.157,E2 -20507.157} C_VEL
LIN {X 0,Y 222.13,Z 759.661,A -85,B 0,C 180,E1 -20510.899,E2 -20510.899} C_VEL
LIN {X 0,Y 222.786,Z 760.598,A -85,B 0,C 180,E1 -20512.752,E2 -20512.752} C_VEL
LIN {X 0,Y 224.518,Z 761.311,A -85,B 0,C 180,E1 -20516.411,E2 -20516.411} C_VEL
LIN {X 0,Y 226.879,Z 760.598,A -85,B 0,C 180,E1 -20520.001,E2 -20520.001} C_VEL
LIN {X 0,Y 229.949,Z 758.437,A -85,B 0,C 180,E1 -20523.505,E2 -20523.505} C_VEL
LIN {X 0,Y 233.66,Z 754.705,A -85,B 0,C 180,E1 -20526.911,E2 -20526.911} C_VEL
LIN {X 0,Y 236.806,Z 750.915,A -85,B 0,C 180,E1 -20529.395,E2 -20529.395} C_VEL
LIN {X 0,Y 240.359,Z 746.074,A -85,B 0,C 180,E1 -20531.811,E2 -20531.811} C_VEL
LIN {X 0,Y 244.942,Z 738.96,A -85,B 0,C 180,E1 -20534.541,E2 -20534.541} C_VEL
LIN {X 0,Y 249.175,Z 731.407,A -85,B 0,C 180,E1 -20536.847,E2 -20536.847} C_VEL
LIN {X 0,Y 253.578,Z 722.551,A -85,B 0,C 180,E1 -20538.996,E2 -20538.996} C_VEL
LIN {X 0,Y 257.85,Z 712.761,A -85,B 0,C 180,E1 -20540.906,E2 -20540.906} C_VEL
LIN {X 0,Y 261.589,Z 702.567,A -85,B 0,C 180,E1 -20542.511,E2 -20542.511} C_VEL
LIN {X 0,Y 265.324,Z 690.624,A -85,B 0,C 180,E1 -20544.033,E2 -20544.033} C_VEL
LIN {X 0,Y 268.32,Z 678.406,A -85,B 0,C 180,E1 -20545.291,E2 -20545.291} C_VEL
LIN {X 0,Y 270.952,Z 663.891,A -85,B 0,C 180,E1 -20546.44,E2 -20546.44} C_VEL
LIN {X 0,Y 272.91,Z 647.903,A -85,B 0,C 180,E1 -20547.35,E2 -20547.35} C_VEL
LIN {X 0,Y 273.998,Z 638.18,A -85,B 0,C 180,E1 -20547.832,E2 -20547.832} C_VEL
LIN {X 0,Y 271.488,Z 632.749,A -85,B 0,C 180,E1 -20549.912,E2 -20549.912} C_VEL
LIN {X 0,Y 269.861,Z 629.663,A -85,B 0,C 180,E1 -20551.58,E2 -20551.58} C_VEL
LIN {X 0,Y 268.68,Z 627.437,A -85,B 0,C 180,E1 -20553.161,E2 -20553.161} C_VEL
LIN {X 0,Y 268.175,Z 626.575,A -85,B 0,C 180,E1 -20553.963,E2 -20553.963} C_VEL
LIN {X 0,Y 267.614,Z 626.531,A -85,B 0,C 180,E1 -20554.791,E2 -20554.791} C_VEL
LIN {X 0,Y 266.511,Z 628.031,A -85,B 0,C 180,E1 -20556.448,E2 -20556.448} C_VEL
LIN {X 0,Y 265.489,Z 631.409,A -85,B 0,C 180,E1 -20559.001,E2 -20559.001} C_VEL
LIN {X 0,Y 265.528,Z 631.998,A -85,B 0,C 180,E1 -20559.877,E2 -20559.877} C_VEL
LIN {X 0,Y 266.534,Z 633.362,A -85,B 0,C 180,E1 -20562.562,E2 -20562.562} C_VEL
LIN {X 0,Y 266.64,Z 634.771,A -85,B 0,C 180,E1 -20563.141,E2 -20563.141} C_VEL
LIN {X 0,Y 266.74,Z 638.974,A -85,B 0,C 180,E1 -20564.218,E2 -20564.218} C_VEL
LIN {X 0,Y 266.695,Z 642.294,A -85,B 0,C 180,E1 -20564.884,E2 -20564.884} C_VEL
LIN {X 0,Y 265.669,Z 657.771,A -85,B 0,C 180,E1 -20566.754,E2 -20566.754} C_VEL
LIN {X 0,Y 264.644,Z 674.024,A -85,B 0,C 180,E1 -20568.403,E2 -20568.403} C_VEL
LIN {X 0,Y 262.115,Z 697.869,A -85,B 0,C 180,E1 -20570.264,E2 -20570.264} C_VEL
LIN {X 0,Y 261.14,Z 702.942,A -85,B 0,C 180,E1 -20570.615,E2 -20570.615} C_VEL
LIN {X 0,Y 256.848,Z 718.619,A -85,B 0,C 180,E1 -20571.628,E2 -20571.628} C_VEL
LIN {X 0,Y 252.351,Z 731.99,A -85,B 0,C 180,E1 -20572.719,E2 -20572.719} C_VEL
LIN {X 0,Y 247.187,Z 744.936,A -85,B 0,C 180,E1 -20574.099,E2 -20574.099} C_VEL
LIN {X 0,Y 241.391,Z 758.001,A -85,B 0,C 180,E1 -20575.914,E2 -20575.914} C_VEL
LIN {X 0,Y 235.634,Z 769.693,A -85,B 0,C 180,E1 -20578.036,E2 -20578.036} C_VEL
LIN {X 0,Y 229.585,Z 781.039,A -85,B 0,C 180,E1 -20580.675,E2 -20580.675} C_VEL
LIN {X 0,Y 224.493,Z 790.231,A -85,B 0,C 180,E1 -20583.507,E2 -20583.507} C_VEL
LIN {X 0,Y 220.283,Z 797.823,A -85,B 0,C 180,E1 -20586.498,E2 -20586.498} C_VEL
LIN {X 0,Y 217.397,Z 803.158,A -85,B 0,C 180,E1 -20589.171,E2 -20589.171} C_VEL
LIN {X 0,Y 215.222,Z 807.549,A -85,B 0,C 180,E1 -20591.929,E2 -20591.929} C_VEL
LIN {X 0,Y 213.71,Z 811.043,A -85,B 0,C 180,E1 -20594.748,E2 -20594.748} C_VEL
LIN {X 0,Y 212.691,Z 814.318,A -85,B 0,C 180,E1 -20598.566,E2 -20598.566} C_VEL
LIN {X 0,Y 212.864,Z 816.127,A -85,B 0,C 180,E1 -20602.412,E2 -20602.412} C_VEL
LIN {X 0,Y 213.244,Z 816.453,A -85,B 0,C 180,E1 -20604.327,E2 -20604.327} C_VEL
LIN {X 0,Y 213.791,Z 816.384,A -85,B 0,C 180,E1 -20606.231,E2 -20606.231} C_VEL
LIN {X 0,Y 214.414,Z 815.862,A -85,B 0,C 180,E1 -20608.123,E2 -20608.123} C_VEL
LIN {X 0,Y 215.146,Z 814.863,A -85,B 0,C 180,E1 -20610.235,E2 -20610.235} C_VEL
LIN {X 0,Y 214.512,Z 815.898,A -85,B 0,C 180,E1 -20611.879,E2 -20611.879} C_VEL
LIN {X 0,Y 213.833,Z 816.674,A -85,B 0,C 180,E1 -20613.77,E2 -20613.77} C_VEL
LIN {X 0,Y 212.837,Z 817.003,A -85,B 0,C 180,E1 -20617.591,E2 -20617.591} C_VEL
LIN {X 0,Y 212.635,Z 815.835,A -85,B 0,C 180,E1 -20621.439,E2 -20621.439} C_VEL
LIN {X 0,Y 213.627,Z 813.275,A -85,B 0,C 180,E1 -20625.26,E2 -20625.26} C_VEL
LIN {X 0,Y 215.709,Z 809.2,A -85,B 0,C 180,E1 -20629.116,E2 -20629.116} C_VEL
LIN {X 0,Y 219.273,Z 803.995,A -85,B 0,C 180,E1 -20632.621,E2 -20632.621} C_VEL
LIN {X 0,Y 224.045,Z 797.169,A -85,B 0,C 180,E1 -20636.052,E2 -20636.052} C_VEL
LIN {X 0,Y 229.899,Z 788.723,A -85,B 0,C 180,E1 -20639.284,E2 -20639.284} C_VEL
LIN {X 0,Y 236.939,Z 778.493,A -85,B 0,C 180,E1 -20642.271,E2 -20642.271} C_VEL
LIN {X 0,Y 242.927,Z 769.401,A -85,B 0,C 180,E1 -20644.344,E2 -20644.344} C_VEL
LIN {X 0,Y 250.709,Z 756.93,A -85,B 0,C 180,E1 -20646.563,E2 -20646.563} C_VEL
LIN {X 0,Y 258.608,Z 743.197,A -85,B 0,C 180,E1 -20648.438,E2 -20648.438} C_VEL
LIN {X 0,Y 265.225,Z 730.507,A -85,B 0,C 180,E1 -20649.784,E2 -20649.784} C_VEL
LIN {X 0,Y 271.961,Z 716.031,A -85,B 0,C 180,E1 -20650.977,E2 -20650.977} C_VEL
LIN {X 0,Y 278.196,Z 700.317,A -85,B 0,C 180,E1 -20652.026,E2 -20652.026} C_VEL
LIN {X 0,Y 284.144,Z 681.299,A -85,B 0,C 180,E1 -20653.354,E2 -20653.354} C_VEL
LIN {X 0,Y 287.1,Z 669.492,A -85,B 0,C 180,E1 -20654.351,E2 -20654.351} C_VEL
LIN {X 0,Y 289.599,Z 658.349,A -85,B 0,C 180,E1 -20655.519,E2 -20655.519} C_VEL
LIN {X 0,Y 289.674,Z 658.042,A -85,B 0,C 180,E1 -20655.676,E2 -20655.676} C_VEL
LIN {X 0,Y 289.873,Z 658.356,A -85,B 0,C 180,E1 -20657.071,E2 -20657.071} C_VEL
LIN {X 0,Y 289.92,Z 659.039,A -85,B 0,C 180,E1 -20657.541,E2 -20657.541} C_VEL
LIN {X 0,Y 286.583,Z 672.956,A -85,B 0,C 180,E1 -20658.536,E2 -20658.536} C_VEL
LIN {X 0,Y 282.476,Z 685.978,A -85,B 0,C 180,E1 -20659.692,E2 -20659.692} C_VEL
LIN {X 0,Y 277.761,Z 698.125,A -85,B 0,C 180,E1 -20660.994,E2 -20660.994} C_VEL
LIN {X 0,Y 272.173,Z 710.297,A -85,B 0,C 180,E1 -20662.64,E2 -20662.64} C_VEL
LIN {X 0,Y 266.243,Z 721.316,A -85,B 0,C 180,E1 -20664.497,E2 -20664.497} C_VEL
LIN {X 0,Y 260.468,Z 730.497,A -85,B 0,C 180,E1 -20666.417,E2 -20666.417} C_VEL
LIN {X 0,Y 254.135,Z 739.497,A -85,B 0,C 180,E1 -20668.766,E2 -20668.766} C_VEL
LIN {X 0,Y 248.125,Z 746.872,A -85,B 0,C 180,E1 -20671.215,E2 -20671.215} C_VEL
LIN {X 0,Y 243.323,Z 752.14,A -85,B 0,C 180,E1 -20673.403,E2 -20673.403} C_VEL
LIN {X 0,Y 237.409,Z 757.752,A -85,B 0,C 180,E1 -20676.444,E2 -20676.444} C_VEL
LIN {X 0,Y 233.382,Z 761.07,A -85,B 0,C 180,E1 -20678.815,E2 -20678.815} C_VEL
LIN {X 0,Y 228.618,Z 764.237,A -85,B 0,C 180,E1 -20682.096,E2 -20682.096} C_VEL
LIN {X 0,Y 224.411,Z 766.229,A -85,B 0,C 180,E1 -20685.49,E2 -20685.49} C_VEL
LIN {X 0,Y 221.168,Z 766.917,A -85,B 0,C 180,E1 -20689.008,E2 -20689.008} C_VEL
LIN {X 0,Y 218.402,Z 766.468,A -85,B 0,C 180,E1 -20692.604,E2 -20692.604} C_VEL
LIN {X 0,Y 216.477,Z 764.781,A -85,B 0,C 180,E1 -20696.276,E2 -20696.276} C_VEL
LIN {X 0,Y 215.152,Z 761.891,A -85,B 0,C 180,E1 -20699.999,E2 -20699.999} C_VEL
LIN {X 0,Y 214.237,Z 757.703,A -85,B 0,C 180,E1 -20703.761,E2 -20703.761} C_VEL
LIN {X 0,Y 214.131,Z 752.114,A -85,B 0,C 180,E1 -20707.543,E2 -20707.543} C_VEL
LIN {X 0,Y 214.34,Z 746.47,A -85,B 0,C 180,E1 -20710.634,E2 -20710.634} C_VEL
LIN {X 0,Y 214.927,Z 738.489,A -85,B 0,C 180,E1 -20714.196,E2 -20714.196} C_VEL
LIN {X 0,Y 215.96,Z 729.352,A -85,B 0,C 180,E1 -20717.518,E2 -20717.518} C_VEL
LIN {X 0,Y 217.173,Z 719.281,A -85,B 0,C 180,E1 -20720.56,E2 -20720.56} C_VEL
LIN {X 0,Y 218.69,Z 707.838,A -85,B 0,C 180,E1 -20723.433,E2 -20723.433} C_VEL
LIN {X 0,Y 220.343,Z 695.46,A -85,B 0,C 180,E1 -20726.011,E2 -20726.011} C_VEL
LIN {X 0,Y 222.033,Z 681.844,A -85,B 0,C 180,E1 -20728.345,E2 -20728.345} C_VEL
LIN {X 0,Y 223.529,Z 668.555,A -85,B 0,C 180,E1 -20730.202,E2 -20730.202} C_VEL
LIN {X 0,Y 225.068,Z 653.03,A -85,B 0,C 180,E1 -20731.93,E2 -20731.93} C_VEL
LIN {X 0,Y 226.231,Z 637.465,A -85,B 0,C 180,E1 -20733.265,E2 -20733.265} C_VEL
LIN {X 0,Y 227.031,Z 621.852,A -85,B 0,C 180,E1 -20734.23,E2 -20734.23} C_VEL
LIN {X 0,Y 227.256,Z 612.683,A -85,B 0,C 180,E1 -20734.702,E2 -20734.702} C_VEL
LIN {X 0,Y 213.799,Z 573.853,A -85,B 0,C 180,E1 -20737.878,E2 -20737.878} C_VEL
LIN {X 0,Y 213.713,Z 573.86,A -85,B 0,C 180,E1 -20741.124,E2 -20741.124} C_VEL
LIN {X 0,Y 213.707,Z 573.863,A -85,B 0,C 180,E1 -20743.677,E2 -20743.677} C_VEL
LIN {X 0,Y 213.709,Z 573.865,A -85,B 0,C 180,E1 -20746.342,E2 -20746.342} C_VEL
LIN {X 0,Y 213.737,Z 573.858,A -85,B 0,C 180,E1 -20751.335,E2 -20751.335} C_VEL
LIN {X 0,Y 213.769,Z 573.855,A -85,B 0,C 180,E1 -20756.019,E2 -20756.019} C_VEL
LIN {X 0,Y 213.76,Z 573.858,A -85,B 0,C 180,E1 -20760.45,E2 -20760.45} C_VEL
LIN {X 0,Y 213.801,Z 573.852,A -85,B 0,C 180,E1 -20764.701,E2 -20764.701} C_VEL
LIN {X 0,Y 213.813,Z 573.852,A -85,B 0,C 180,E1 -20768.802,E2 -20768.802} C_VEL
LIN {X 0,Y 213.943,Z 573.836,A -85,B 0,C 180,E1 -20772.802,E2 -20772.802} C_VEL
LIN {X 0,Y 213.98,Z 573.828,A -85,B 0,C 180,E1 -20776.707,E2 -20776.707} C_VEL
LIN {X 0,Y 214.195,Z 573.803,A -85,B 0,C 180,E1 -20780.557,E2 -20780.557} C_VEL
LIN {X 0,Y 214.247,Z 573.795,A -85,B 0,C 180,E1 -20782.459,E2 -20782.459} C_VEL
LIN {X 0,Y 214.445,Z 573.771,A -85,B 0,C 180,E1 -20788.121,E2 -20788.121} C_VEL
LIN {X 0,Y 214.549,Z 573.757,A -85,B 0,C 180,E1 -20789.999,E2 -20789.999} C_VEL
LIN {X 0,Y 214.444,Z 573.768,A -85,B 0,C 180,E1 -20791.877,E2 -20791.877} C_VEL
LIN {X 0,Y 214.245,Z 573.798,A -85,B 0,C 180,E1 -20797.539,E2 -20797.539} C_VEL
LIN {X 0,Y 214.045,Z 573.82,A -85,B 0,C 180,E1 -20801.361,E2 -20801.361} C_VEL
LIN {X 0,Y 213.931,Z 573.837,A -85,B 0,C 180,E1 -20805.236,E2 -20805.236} C_VEL
LIN {X 0,Y 213.873,Z 573.843,A -85,B 0,C 180,E1 -20809.183,E2 -20809.183} C_VEL
LIN {X 0,Y 213.852,Z 573.845,A -85,B 0,C 180,E1 -20813.225,E2 -20813.225} C_VEL
LIN {X 0,Y 213.825,Z 573.85,A -85,B 0,C 180,E1 -20817.449,E2 -20817.449} C_VEL
LIN {X 0,Y 213.775,Z 573.856,A -85,B 0,C 180,E1 -20821.735,E2 -20821.735} C_VEL
LIN {X 0,Y 213.75,Z 573.859,A -85,B 0,C 180,E1 -20826.286,E2 -20826.286} C_VEL
LIN {X 0,Y 213.786,Z 573.853,A -85,B 0,C 180,E1 -20831.106,E2 -20831.106} C_VEL
LIN {X 0,Y 213.816,Z 573.851,A -85,B 0,C 180,E1 -20834.311,E2 -20834.311} C_VEL
LIN {X 0,Y 226.575,Z 609.454,A -85,B 0,C 180,E1 -20837.124,E2 -20837.124} C_VEL
LIN {X 0,Y 225.416,Z 642.854,A -85,B 0,C 180,E1 -20838.735,E2 -20838.735} C_VEL
LIN {X 0,Y 224.576,Z 657.283,A -85,B 0,C 180,E1 -20839.802,E2 -20839.802} C_VEL
LIN {X 0,Y 223.346,Z 671.352,A -85,B 0,C 180,E1 -20841.198,E2 -20841.198} C_VEL
LIN {X 0,Y 221.987,Z 684.284,A -85,B 0,C 180,E1 -20842.846,E2 -20842.846} C_VEL
LIN {X 0,Y 220.374,Z 697.456,A -85,B 0,C 180,E1 -20844.968,E2 -20844.968} C_VEL
LIN {X 0,Y 218.893,Z 708.713,A -85,B 0,C 180,E1 -20847.194,E2 -20847.194} C_VEL
LIN {X 0,Y 217.607,Z 718.1,A -85,B 0,C 180,E1 -20849.425,E2 -20849.425} C_VEL
LIN {X 0,Y 216.42,Z 726.892,A -85,B 0,C 180,E1 -20851.91,E2 -20851.91} C_VEL
LIN {X 0,Y 215.328,Z 735.662,A -85,B 0,C 180,E1 -20854.895,E2 -20854.895} C_VEL
LIN {X 0,Y 214.563,Z 742.767,A -85,B 0,C 180,E1 -20857.873,E2 -20857.873} C_VEL
LIN {X 0,Y 214.096,Z 748.563,A -85,B 0,C 180,E1 -20860.837,E2 -20860.837} C_VEL
LIN {X 0,Y 213.984,Z 753.225,A -85,B 0,C 180,E1 -20863.79,E2 -20863.79} C_VEL
LIN {X 0,Y 214.217,Z 756.849,A -85,B 0,C 180,E1 -20866.724,E2 -20866.724} C_VEL
LIN {X 0,Y 214.648,Z 759.175,A -85,B 0,C 180,E1 -20869.184,E2 -20869.184} C_VEL
LIN {X 0,Y 215.644,Z 761.366,A -85,B 0,C 180,E1 -20872.51,E2 -20872.51} C_VEL
LIN {X 0,Y 217.397,Z 762.518,A -85,B 0,C 180,E1 -20876.294,E2 -20876.294} C_VEL
LIN {X 0,Y 219.823,Z 762.23,A -85,B 0,C 180,E1 -20880.001,E2 -20880.001} C_VEL
LIN {X 0,Y 222.983,Z 760.435,A -85,B 0,C 180,E1 -20883.615,E2 -20883.615} C_VEL
LIN {X 0,Y 226.818,Z 757.186,A -85,B 0,C 180,E1 -20887.12,E2 -20887.12} C_VEL
LIN {X 0,Y 230.064,Z 753.713,A -85,B 0,C 180,E1 -20889.673,E2 -20889.673} C_VEL
LIN {X 0,Y 235.084,Z 747.589,A -85,B 0,C 180,E1 -20892.958,E2 -20892.958} C_VEL
LIN {X 0,Y 239.974,Z 740.542,A -85,B 0,C 180,E1 -20895.719,E2 -20895.719} C_VEL
LIN {X 0,Y 245.184,Z 731.87,A -85,B 0,C 180,E1 -20898.38,E2 -20898.38} C_VEL
LIN {X 0,Y 250.023,Z 722.611,A -85,B 0,C 180,E1 -20900.572,E2 -20900.572} C_VEL
LIN {X 0,Y 255.057,Z 711.345,A -85,B 0,C 180,E1 -20902.692,E2 -20902.692} C_VEL
LIN {X 0,Y 258.986,Z 700.995,A -85,B 0,C 180,E1 -20904.233,E2 -20904.233} C_VEL
LIN {X 0,Y 262.897,Z 688.41,A -85,B 0,C 180,E1 -20905.748,E2 -20905.748} C_VEL
LIN {X 0,Y 266.061,Z 675.273,A -85,B 0,C 180,E1 -20907.016,E2 -20907.016} C_VEL
LIN {X 0,Y 268.463,Z 661.489,A -85,B 0,C 180,E1 -20908.012,E2 -20908.012} C_VEL
LIN {X 0,Y 270.857,Z 642.467,A -85,B 0,C 180,E1 -20909.046,E2 -20909.046} C_VEL
LIN {X 0,Y 268.899,Z 638.122,A -85,B 0,C 180,E1 -20910.938,E2 -20910.938} C_VEL
LIN {X 0,Y 267.95,Z 636.19,A -85,B 0,C 180,E1 -20912.048,E2 -20912.048} C_VEL
LIN {X 0,Y 266.668,Z 633.214,A -85,B 0,C 180,E1 -20914.089,E2 -20914.089} C_VEL
LIN {X 0,Y 265.437,Z 631.791,A -85,B 0,C 180,E1 -20917.411,E2 -20917.411} C_VEL
LIN {X 0,Y 265.528,Z 631.998,A -85,B 0,C 180,E1 -20919.877,E2 -20919.877} C_VEL
LIN {X 0,Y 265.592,Z 633.015,A -85,B 0,C 180,E1 -20920.696,E2 -20920.696} C_VEL
LIN {X 0,Y 265.414,Z 635.912,A -85,B 0,C 180,E1 -20921.657,E2 -20921.657} C_VEL
LIN {X 0,Y 264.992,Z 640.919,A -85,B 0,C 180,E1 -20922.697,E2 -20922.697} C_VEL
LIN {X 0,Y 264.672,Z 645.208,A -85,B 0,C 180,E1 -20923.484,E2 -20923.484} C_VEL
LIN {X 0,Y 264.442,Z 648.247,A -85,B 0,C 180,E1 -20923.943,E2 -20923.943} C_VEL
LIN {X 0,Y 263.226,Z 661.421,A -85,B 0,C 180,E1 -20925.525,E2 -20925.525} C_VEL
LIN {X 0,Y 261.969,Z 676.292,A -85,B 0,C 180,E1 -20927.061,E2 -20927.061} C_VEL
LIN {X 0,Y 259.391,Z 696.208,A -85,B 0,C 180,E1 -20928.646,E2 -20928.646} C_VEL
LIN {X 0,Y 258.064,Z 702.95,A -85,B 0,C 180,E1 -20929.188,E2 -20929.188} C_VEL
LIN {X 0,Y 253.707,Z 717.926,A -85,B 0,C 180,E1 -20930.165,E2 -20930.165} C_VEL
LIN {X 0,Y 248.697,Z 731.701,A -85,B 0,C 180,E1 -20931.302,E2 -20931.302} C_VEL
LIN {X 0,Y 242.733,Z 745.617,A -85,B 0,C 180,E1 -20932.815,E2 -20932.815} C_VEL
LIN {X 0,Y 236.691,Z 758.171,A -85,B 0,C 180,E1 -20934.621,E2 -20934.621} C_VEL
LIN {X 0,Y 230.658,Z 769.523,A -85,B 0,C 180,E1 -20936.741,E2 -20936.741} C_VEL
LIN {X 0,Y 225.22,Z 779.087,A -85,B 0,C 180,E1 -20939.012,E2 -20939.012} C_VEL
LIN {X 0,Y 219.582,Z 788.347,A -85,B 0,C 180,E1 -20941.831,E2 -20941.831} C_VEL
LIN {X 0,Y 214.951,Z 795.949,A -85,B 0,C 180,E1 -20944.848,E2 -20944.848} C_VEL
LIN {X 0,Y 211.677,Z 801.351,A -85,B 0,C 180,E1 -20947.555,E2 -20947.555} C_VEL
LIN {X 0,Y 209.08,Z 805.795,A -85,B 0,C 180,E1 -20950.359,E2 -20950.359} C_VEL
LIN {X 0,Y 206.813,Z 810.326,A -85,B 0,C 180,E1 -20954.226,E2 -20954.226} C_VEL
LIN {X 0,Y 205.674,Z 813.38,A -85,B 0,C 180,E1 -20958.17,E2 -20958.17} C_VEL
LIN {X 0,Y 205.783,Z 814.98,A -85,B 0,C 180,E1 -20962.149,E2 -20962.149} C_VEL
LIN {X 0,Y 206.19,Z 815.187,A -85,B 0,C 180,E1 -20964.132,E2 -20964.132} C_VEL
LIN {X 0,Y 206.771,Z 814.99,A -85,B 0,C 180,E1 -20966.103,E2 -20966.103} C_VEL
LIN {X 0,Y 207.428,Z 814.377,A -85,B 0,C 180,E1 -20968.06,E2 -20968.06} C_VEL
LIN {X 0,Y 208.182,Z 813.164,A -85,B 0,C 180,E1 -20970.364,E2 -20970.364} C_VEL
LIN {X 0,Y 207.593,Z 814.21,A -85,B 0,C 180,E1 -20971.941,E2 -20971.941} C_VEL
LIN {X 0,Y 206.861,Z 815.078,A -85,B 0,C 180,E1 -20973.897,E2 -20973.897} C_VEL
LIN {X 0,Y 205.804,Z 815.605,A -85,B 0,C 180,E1 -20977.973,E2 -20977.973} C_VEL
LIN {X 0,Y 205.658,Z 814.692,A -85,B 0,C 180,E1 -20981.833,E2 -20981.833} C_VEL
LIN {X 0,Y 206.729,Z 812.419,A -85,B 0,C 180,E1 -20985.783,E2 -20985.783} C_VEL
LIN {X 0,Y 208.923,Z 808.798,A -85,B 0,C 180,E1 -20989.658,E2 -20989.658} C_VEL
LIN {X 0,Y 212.718,Z 803.862,A -85,B 0,C 180,E1 -20993.359,E2 -20993.359} C_VEL
LIN {X 0,Y 217.703,Z 797.501,A -85,B 0,C 180,E1 -20996.87,E2 -20996.87} C_VEL
LIN {X 0,Y 223.791,Z 789.609,A -85,B 0,C 180,E1 -21000.165,E2 -21000.165} C_VEL
LIN {X 0,Y 231.063,Z 779.993,A -85,B 0,C 180,E1 -21003.196,E2 -21003.196} C_VEL
LIN {X 0,Y 238.318,Z 769.96,A -85,B 0,C 180,E1 -21005.623,E2 -21005.623} C_VEL
LIN {X 0,Y 246.39,Z 758.136,A -85,B 0,C 180,E1 -21007.827,E2 -21007.827} C_VEL
LIN {X 0,Y 254.548,Z 745.186,A -85,B 0,C 180,E1 -21009.679,E2 -21009.679} C_VEL
LIN {X 0,Y 261.893,Z 732.298,A -85,B 0,C 180,E1 -21011.095,E2 -21011.095} C_VEL
LIN {X 0,Y 269.735,Z 716.794,A -85,B 0,C 180,E1 -21012.391,E2 -21012.391} C_VEL
LIN {X 0,Y 276.626,Z 700.891,A -85,B 0,C 180,E1 -21013.473,E2 -21013.473} C_VEL
LIN {X 0,Y 283.057,Z 682.526,A -85,B 0,C 180,E1 -21014.766,E2 -21014.766} C_VEL
LIN {X 0,Y 286.339,Z 671.448,A -85,B 0,C 180,E1 -21015.723,E2 -21015.723} C_VEL
LIN {X 0,Y 287.912,Z 665.695,A -85,B 0,C 180,E1 -21016.295,E2 -21016.295} C_VEL
LIN {X 0,Y 287.918,Z 665.826,A -85,B 0,C 180,E1 -21016.533,E2 -21016.533} C_VEL
LIN {X 0,Y 284.037,Z 679.32,A -85,B 0,C 180,E1 -21017.541,E2 -21017.541} C_VEL
LIN {X 0,Y 279.03,Z 693.042,A -85,B 0,C 180,E1 -21018.85,E2 -21018.85} C_VEL
LIN {X 0,Y 274.629,Z 703.047,A -85,B 0,C 180,E1 -21019.986,E2 -21019.986} C_VEL
LIN {X 0,Y 268.75,Z 714.486,A -85,B 0,C 180,E1 -21021.604,E2 -21021.604} C_VEL
LIN {X 0,Y 262.398,Z 725.12,A -85,B 0,C 180,E1 -21023.468,E2 -21023.468} C_VEL
LIN {X 0,Y 256.463,Z 733.861,A -85,B 0,C 180,E1 -21025.345,E2 -21025.345} C_VEL
LIN {X 0,Y 249.774,Z 742.423,A -85,B 0,C 180,E1 -21027.682,E2 -21027.682} C_VEL
LIN {X 0,Y 244.341,Z 748.607,A -85,B 0,C 180,E1 -21029.777,E2 -21029.777} C_VEL
LIN {X 0,Y 237.576,Z 755.315,A -85,B 0,C 180,E1 -21032.707,E2 -21032.707} C_VEL
LIN {X 0,Y 231.388,Z 760.531,A -85,B 0,C 180,E1 -21035.792,E2 -21035.792} C_VEL
LIN {X 0,Y 227.165,Z 763.481,A -85,B 0,C 180,E1 -21038.206,E2 -21038.206} C_VEL
LIN {X 0,Y 222.175,Z 766.339,A -85,B 0,C 180,E1 -21041.558,E2 -21041.558} C_VEL
LIN {X 0,Y 217.769,Z 767.954,A -85,B 0,C 180,E1 -21045.037,E2 -21045.037} C_VEL
LIN {X 0,Y 214.368,Z 768.34,A -85,B 0,C 180,E1 -21048.655,E2 -21048.655} C_VEL
LIN {X 0,Y 211.461,Z 767.566,A -85,B 0,C 180,E1 -21052.36,E2 -21052.36} C_VEL
LIN {X 0,Y 209.45,Z 765.575,A -85,B 0,C 180,E1 -21056.151,E2 -21056.151} C_VEL
LIN {X 0,Y 208.054,Z 762.374,A -85,B 0,C 180,E1 -21059.999,E2 -21059.999} C_VEL
LIN {X 0,Y 207.139,Z 757.888,A -85,B 0,C 180,E1 -21063.89,E2 -21063.89} C_VEL
LIN {X 0,Y 207.062,Z 751.978,A -85,B 0,C 180,E1 -21067.802,E2 -21067.802} C_VEL
LIN {X 0,Y 207.399,Z 744.49,A -85,B 0,C 180,E1 -21071.73,E2 -21071.73} C_VEL
LIN {X 0,Y 208.038,Z 736.389,A -85,B 0,C 180,E1 -21075.177,E2 -21075.177} C_VEL
LIN {X 0,Y 209.195,Z 726.585,A -85,B 0,C 180,E1 -21078.611,E2 -21078.611} C_VEL
LIN {X 0,Y 210.47,Z 716.522,A -85,B 0,C 180,E1 -21081.549,E2 -21081.549} C_VEL
LIN {X 0,Y 212.15,Z 704.449,A -85,B 0,C 180,E1 -21084.461,E2 -21084.461} C_VEL
LIN {X 0,Y 213.889,Z 691.084,A -85,B 0,C 180,E1 -21087.122,E2 -21087.122} C_VEL
LIN {X 0,Y 215.517,Z 677.846,A -85,B 0,C 180,E1 -21089.284,E2 -21089.284} C_VEL
LIN {X 0,Y 217.111,Z 663.352,A -85,B 0,C 180,E1 -21091.192,E2 -21091.192} C_VEL
LIN {X 0,Y 218.467,Z 648.453,A -85,B 0,C 180,E1 -21092.741,E2 -21092.741} C_VEL
LIN {X 0,Y 219.567,Z 632.568,A -85,B 0,C 180,E1 -21093.993,E2 -21093.993} C_VEL
LIN {X 0,Y 220.287,Z 614.049,A -85,B 0,C 180,E1 -21095.057,E2 -21095.057} C_VEL
LIN {X 0,Y 206.745,Z 574.732,A -85,B 0,C 180,E1 -21098.396,E2 -21098.396} C_VEL
LIN {X 0,Y 206.625,Z 574.745,A -85,B 0,C 180,E1 -21102.863,E2 -21102.863} C_VEL
LIN {X 0,Y 206.628,Z 574.742,A -85,B 0,C 180,E1 -21107.135,E2 -21107.135} C_VEL
LIN {X 0,Y 206.702,Z 574.735,A -85,B 0,C 180,E1 -21111.444,E2 -21111.444} C_VEL
LIN {X 0,Y 206.732,Z 574.733,A -85,B 0,C 180,E1 -21114.694,E2 -21114.694} C_VEL
LIN {X 0,Y 206.707,Z 574.734,A -85,B 0,C 180,E1 -21119.335,E2 -21119.335} C_VEL
LIN {X 0,Y 206.732,Z 574.731,A -85,B 0,C 180,E1 -21123.771,E2 -21123.771} C_VEL
LIN {X 0,Y 206.757,Z 574.726,A -85,B 0,C 180,E1 -21128.042,E2 -21128.042} C_VEL
LIN {X 0,Y 206.876,Z 574.714,A -85,B 0,C 180,E1 -21132.196,E2 -21132.196} C_VEL
LIN {X 0,Y 206.913,Z 574.706,A -85,B 0,C 180,E1 -21136.244,E2 -21136.244} C_VEL
LIN {X 0,Y 207.131,Z 574.682,A -85,B 0,C 180,E1 -21140.231,E2 -21140.231} C_VEL
LIN {X 0,Y 207.187,Z 574.674,A -85,B 0,C 180,E1 -21142.201,E2 -21142.201} C_VEL
LIN {X 0,Y 207.381,Z 574.651,A -85,B 0,C 180,E1 -21148.057,E2 -21148.057} C_VEL
LIN {X 0,Y 207.513,Z 574.634,A -85,B 0,C 180,E1 -21149.999,E2 -21149.999} C_VEL
LIN {X 0,Y 207.381,Z 574.648,A -85,B 0,C 180,E1 -21151.941,E2 -21151.941} C_VEL
LIN {X 0,Y 207.186,Z 574.676,A -85,B 0,C 180,E1 -21157.797,E2 -21157.797} C_VEL
LIN {X 0,Y 206.981,Z 574.698,A -85,B 0,C 180,E1 -21161.754,E2 -21161.754} C_VEL
LIN {X 0,Y 206.865,Z 574.717,A -85,B 0,C 180,E1 -21165.77,E2 -21165.77} C_VEL
LIN {X 0,Y 206.809,Z 574.72,A -85,B 0,C 180,E1 -21169.865,E2 -21169.865} C_VEL
LIN {X 0,Y 206.764,Z 574.729,A -85,B 0,C 180,E1 -21174.071,E2 -21174.071} C_VEL
LIN {X 0,Y 206.74,Z 574.728,A -85,B 0,C 180,E1 -21178.418,E2 -21178.418} C_VEL
LIN {X 0,Y 206.705,Z 574.735,A -85,B 0,C 180,E1 -21182.955,E2 -21182.955} C_VEL
LIN {X 0,Y 206.72,Z 574.737,A -85,B 0,C 180,E1 -21187.73,E2 -21187.73} C_VEL
LIN {X 0,Y 206.717,Z 574.736,A -85,B 0,C 180,E1 -21191.587,E2 -21191.587} C_VEL
LIN {X 0,Y 206.804,Z 574.883,A -85,B 0,C 180,E1 -21193.738,E2 -21193.738} C_VEL
LIN {X 0,Y 219.684,Z 611.013,A -85,B 0,C 180,E1 -21196.701,E2 -21196.701} C_VEL
LIN {X 0,Y 218.48,Z 644.02,A -85,B 0,C 180,E1 -21198.36,E2 -21198.36} C_VEL
LIN {X 0,Y 217.611,Z 658.449,A -85,B 0,C 180,E1 -21199.463,E2 -21199.463} C_VEL
LIN {X 0,Y 216.353,Z 672.568,A -85,B 0,C 180,E1 -21200.911,E2 -21200.911} C_VEL
LIN {X 0,Y 215.018,Z 684.726,A -85,B 0,C 180,E1 -21202.501,E2 -21202.501} C_VEL
LIN {X 0,Y 213.452,Z 697.206,A -85,B 0,C 180,E1 -21204.53,E2 -21204.53} C_VEL
LIN {X 0,Y 211.95,Z 708.69,A -85,B 0,C 180,E1 -21206.831,E2 -21206.831} C_VEL
LIN {X 0,Y 210.471,Z 719.183,A -85,B 0,C 180,E1 -21209.389,E2 -21209.389} C_VEL
LIN {X 0,Y 209.279,Z 727.951,A -85,B 0,C 180,E1 -21211.957,E2 -21211.957} C_VEL
LIN {X 0,Y 208.197,Z 736.704,A -85,B 0,C 180,E1 -21215.04,E2 -21215.04} C_VEL
LIN {X 0,Y 207.424,Z 743.846,A -85,B 0,C 180,E1 -21218.118,E2 -21218.118} C_VEL
LIN {X 0,Y 206.914,Z 750.999,A -85,B 0,C 180,E1 -21221.993,E2 -21221.993} C_VEL
LIN {X 0,Y 206.979,Z 755.668,A -85,B 0,C 180,E1 -21225.247,E2 -21225.247} C_VEL
LIN {X 0,Y 207.558,Z 759.772,A -85,B 0,C 180,E1 -21229.091,E2 -21229.091} C_VEL
LIN {X 0,Y 208.467,Z 762.061,A -85,B 0,C 180,E1 -21232.251,E2 -21232.251} C_VEL
LIN {X 0,Y 210.263,Z 763.629,A -85,B 0,C 180,E1 -21236.168,E2 -21236.168} C_VEL
LIN {X 0,Y 212.729,Z 763.715,A -85,B 0,C 180,E1 -21240.001,E2 -21240.001} C_VEL
LIN {X 0,Y 216.005,Z 762.377,A -85,B 0,C 180,E1 -21243.732,E2 -21243.732} C_VEL
LIN {X 0,Y 219.973,Z 759.571,A -85,B 0,C 180,E1 -21247.343,E2 -21247.343} C_VEL
LIN {X 0,Y 224.58,Z 755.214,A -85,B 0,C 180,E1 -21250.823,E2 -21250.823} C_VEL
LIN {X 0,Y 228.531,Z 750.828,A -85,B 0,C 180,E1 -21253.336,E2 -21253.336} C_VEL
LIN {X 0,Y 233.616,Z 744.374,A -85,B 0,C 180,E1 -21256.158,E2 -21256.158} C_VEL
LIN {X 0,Y 239.059,Z 736.318,A -85,B 0,C 180,E1 -21258.869,E2 -21258.869} C_VEL
LIN {X 0,Y 244.064,Z 727.808,A -85,B 0,C 180,E1 -21261.098,E2 -21261.098} C_VEL
LIN {X 0,Y 249.329,Z 717.403,A -85,B 0,C 180,E1 -21263.243,E2 -21263.243} C_VEL
LIN {X 0,Y 253.88,Z 706.974,A -85,B 0,C 180,E1 -21264.972,E2 -21264.972} C_VEL
LIN {X 0,Y 258.478,Z 694.03,A -85,B 0,C 180,E1 -21266.657,E2 -21266.657} C_VEL
LIN {X 0,Y 262.124,Z 681.225,A -85,B 0,C 180,E1 -21267.983,E2 -21267.983} C_VEL
LIN {X 0,Y 264.965,Z 667.786,A -85,B 0,C 180,E1 -21269.065,E2 -21269.065} C_VEL
LIN {X 0,Y 267.36,Z 651.368,A -85,B 0,C 180,E1 -21270.032,E2 -21270.032} C_VEL
LIN {X 0,Y 267.924,Z 646.976,A -85,B 0,C 180,E1 -21270.29,E2 -21270.29} C_VEL
LIN {X 0,Y 266.391,Z 643.212,A -85,B 0,C 180,E1 -21272.121,E2 -21272.121} C_VEL
LIN {X 0,Y 264.966,Z 639.942,A -85,B 0,C 180,E1 -21274.494,E2 -21274.494} C_VEL
LIN {X 0,Y 264.056,Z 638.793,A -85,B 0,C 180,E1 -21277.018,E2 -21277.018} C_VEL
LIN {X 0,Y 264.021,Z 638.912,A -85,B 0,C 180,E1 -21279.783,E2 -21279.783} C_VEL
LIN {X 0,Y 264.836,Z 640.207,A -85,B 0,C 180,E1 -21282.237,E2 -21282.237} C_VEL
LIN {X 0,Y 264.691,Z 644.67,A -85,B 0,C 180,E1 -21283.377,E2 -21283.377} C_VEL
LIN {X 0,Y 264.672,Z 645.208,A -85,B 0,C 180,E1 -21283.484,E2 -21283.484} C_VEL
LIN {X 0,Y 264.382,Z 648.021,A -85,B 0,C 180,E1 -21283.829,E2 -21283.829} C_VEL
LIN {X 0,Y 263.567,Z 652.535,A -85,B 0,C 180,E1 -21284.008,E2 -21284.008} C_VEL
LIN {X 0,Y 261.573,Z 661.972,A -85,B 0,C 180,E1 -21284.079,E2 -21284.079} C_VEL
LIN {X 0,Y 261.002,Z 665.807,A -85,B 0,C 180,E1 -21284.353,E2 -21284.353} C_VEL
LIN {X 0,Y 259.536,Z 679.156,A -85,B 0,C 180,E1 -21285.722,E2 -21285.722} C_VEL
LIN {X 0,Y 256.992,Z 695.087,A -85,B 0,C 180,E1 -21287.031,E2 -21287.031} C_VEL
LIN {X 0,Y 255.219,Z 703.341,A -85,B 0,C 180,E1 -21287.734,E2 -21287.734} C_VEL
LIN {X 0,Y 251.105,Z 716.608,A -85,B 0,C 180,E1 -21288.608,E2 -21288.608} C_VEL
LIN {X 0,Y 245.855,Z 730.156,A -85,B 0,C 180,E1 -21289.704,E2 -21289.704} C_VEL
LIN {X 0,Y 239.664,Z 743.985,A -85,B 0,C 180,E1 -21291.186,E2 -21291.186} C_VEL
LIN {X 0,Y 233.824,Z 755.412,A -85,B 0,C 180,E1 -21292.78,E2 -21292.78} C_VEL
LIN {X 0,Y 226.85,Z 767.765,A -85,B 0,C 180,E1 -21295.032,E2 -21295.032} C_VEL
LIN {X 0,Y 221.056,Z 777.254,A -85,B 0,C 180,E1 -21297.285,E2 -21297.285} C_VEL
LIN {X 0,Y 215.812,Z 785.352,A -85,B 0,C 180,E1 -21299.686,E2 -21299.686} C_VEL
LIN {X 0,Y 210.52,Z 793.182,A -85,B 0,C 180,E1 -21302.677,E2 -21302.677} C_VEL
LIN {X 0,Y 206.164,Z 799.598,A -85,B 0,C 180,E1 -21305.855,E2 -21305.855} C_VEL
LIN {X 0,Y 202.354,Z 805.366,A -85,B 0,C 180,E1 -21309.678,E2 -21309.678} C_VEL
LIN {X 0,Y 199.935,Z 809.631,A -85,B 0,C 180,E1 -21313.669,E2 -21313.669} C_VEL
LIN {X 0,Y 198.68,Z 812.403,A -85,B 0,C 180,E1 -21317.748,E2 -21317.748} C_VEL
LIN {X 0,Y 198.751,Z 813.748,A -85,B 0,C 180,E1 -21321.938,E2 -21321.938} C_VEL
LIN {X 0,Y 199.761,Z 813.586,A -85,B 0,C 180,E1 -21325.966,E2 -21325.966} C_VEL
LIN {X 0,Y 200.458,Z 812.896,A -85,B 0,C 180,E1 -21327.992,E2 -21327.992} C_VEL
LIN {X 0,Y 201.313,Z 811.389,A -85,B 0,C 180,E1 -21330.439,E2 -21330.439} C_VEL
LIN {X 0,Y 199.909,Z 813.425,A -85,B 0,C 180,E1 -21334.033,E2 -21334.033} C_VEL
LIN {X 0,Y 198.808,Z 814.2,A -85,B 0,C 180,E1 -21338.177,E2 -21338.177} C_VEL
LIN {X 0,Y 198.698,Z 813.539,A -85,B 0,C 180,E1 -21342.254,E2 -21342.254} C_VEL
LIN {X 0,Y 199.856,Z 811.555,A -85,B 0,C 180,E1 -21346.34,E2 -21346.34} C_VEL
LIN {X 0,Y 202.223,Z 808.269,A -85,B 0,C 180,E1 -21350.338,E2 -21350.338} C_VEL
LIN {X 0,Y 206.194,Z 803.71,A -85,B 0,C 180,E1 -21354.144,E2 -21354.144} C_VEL
LIN {X 0,Y 211.396,Z 797.788,A -85,B 0,C 180,E1 -21357.74,E2 -21357.74} C_VEL
LIN {X 0,Y 217.737,Z 790.393,A -85,B 0,C 180,E1 -21361.095,E2 -21361.095} C_VEL
LIN {X 0,Y 225.247,Z 781.415,A -85,B 0,C 180,E1 -21364.169,E2 -21364.169} C_VEL
LIN {X 0,Y 232.695,Z 772.08,A -85,B 0,C 180,E1 -21366.621,E2 -21366.621} C_VEL
LIN {X 0,Y 240.962,Z 761.112,A -85,B 0,C 180,E1 -21368.836,E2 -21368.836} C_VEL
LIN {X 0,Y 248.618,Z 750.156,A -85,B 0,C 180,E1 -21370.555,E2 -21370.555} C_VEL
LIN {X 0,Y 257.447,Z 736.313,A -85,B 0,C 180,E1 -21372.228,E2 -21372.228} C_VEL
LIN {X 0,Y 265.471,Z 722.161,A -85,B 0,C 180,E1 -21373.498,E2 -21373.498} C_VEL
LIN {X 0,Y 273.737,Z 705.405,A -85,B 0,C 180,E1 -21374.656,E2 -21374.656} C_VEL
LIN {X 0,Y 281.383,Z 686.412,A -85,B 0,C 180,E1 -21375.989,E2 -21375.989} C_VEL
LIN {X 0,Y 282.385,Z 683.652,A -85,B 0,C 180,E1 -21376.2,E2 -21376.2} C_VEL
LIN {X 0,Y 281.876,Z 684.987,A -85,B 0,C 180,E1 -21376.492,E2 -21376.492} C_VEL
LIN {X 0,Y 276.168,Z 698.732,A -85,B 0,C 180,E1 -21377.84,E2 -21377.84} C_VEL
LIN {X 0,Y 269.929,Z 711.095,A -85,B 0,C 180,E1 -21379.389,E2 -21379.389} C_VEL
LIN {X 0,Y 264.351,Z 720.583,A -85,B 0,C 180,E1 -21380.845,E2 -21380.845} C_VEL
LIN {X 0,Y 256.731,Z 731.75,A -85,B 0,C 180,E1 -21382.968,E2 -21382.968} C_VEL
LIN {X 0,Y 249.523,Z 740.955,A -85,B 0,C 180,E1 -21385.224,E2 -21385.224} C_VEL
LIN {X 0,Y 243.615,Z 747.545,A -85,B 0,C 180,E1 -21387.253,E2 -21387.253} C_VEL
LIN {X 0,Y 237.067,Z 753.949,A -85,B 0,C 180,E1 -21389.736,E2 -21389.736} C_VEL
LIN {X 0,Y 230.15,Z 759.796,A -85,B 0,C 180,E1 -21392.738,E2 -21392.738} C_VEL
LIN {X 0,Y 223.862,Z 764.208,A -85,B 0,C 180,E1 -21395.912,E2 -21395.912} C_VEL
LIN {X 0,Y 218.253,Z 767.294,A -85,B 0,C 180,E1 -21399.254,E2 -21399.254} C_VEL
LIN {X 0,Y 213.339,Z 769.176,A -85,B 0,C 180,E1 -21402.752,E2 -21402.752} C_VEL
LIN {X 0,Y 209.165,Z 769.855,A -85,B 0,C 180,E1 -21406.396,E2 -21406.396} C_VEL
LIN {X 0,Y 205.947,Z 769.325,A -85,B 0,C 180,E1 -21410.175,E2 -21410.175} C_VEL
LIN {X 0,Y 203.404,Z 767.628,A -85,B 0,C 180,E1 -21414.049,E2 -21414.049} C_VEL
LIN {X 0,Y 201.593,Z 764.738,A -85,B 0,C 180,E1 -21418.001,E2 -21418.001} C_VEL
LIN {X 0,Y 200.426,Z 760.571,A -85,B 0,C 180,E1 -21422.009,E2 -21422.009} C_VEL
LIN {X 0,Y 199.937,Z 755.041,A -85,B 0,C 180,E1 -21426.052,E2 -21426.052} C_VEL
LIN {X 0,Y 200.075,Z 749.924,A -85,B 0,C 180,E1 -21429.094,E2 -21429.094} C_VEL
LIN {X 0,Y 200.43,Z 742.71,A -85,B 0,C 180,E1 -21432.658,E2 -21432.658} C_VEL
LIN {X 0,Y 201.22,Z 733.965,A -85,B 0,C 180,E1 -21436.224,E2 -21436.224} C_VEL
LIN {X 0,Y 202.352,Z 725.031,A -85,B 0,C 180,E1 -21439.265,E2 -21439.265} C_VEL
LIN {X 0,Y 203.737,Z 714.46,A -85,B 0,C 180,E1 -21442.299,E2 -21442.299} C_VEL
LIN {X 0,Y 205.339,Z 702.961,A -85,B 0,C 180,E1 -21445.058,E2 -21445.058} C_VEL
LIN {X 0,Y 206.991,Z 690.455,A -85,B 0,C 180,E1 -21447.555,E2 -21447.555} C_VEL
LIN {X 0,Y 208.684,Z 676.829,A -85,B 0,C 180,E1 -21449.784,E2 -21449.784} C_VEL
LIN {X 0,Y 210.341,Z 661.803,A -85,B 0,C 180,E1 -21451.751,E2 -21451.751} C_VEL
LIN {X 0,Y 211.731,Z 646.207,A -85,B 0,C 180,E1 -21453.35,E2 -21453.35} C_VEL
LIN {X 0,Y 212.768,Z 630.758,A -85,B 0,C 180,E1 -21454.526,E2 -21454.526} C_VEL
LIN {X 0,Y 213.378,Z 615.46,A -85,B 0,C 180,E1 -21455.405,E2 -21455.405} C_VEL
LIN {X 0,Y 199.688,Z 575.609,A -85,B 0,C 180,E1 -21458.918,E2 -21458.918} C_VEL
LIN {X 0,Y 199.575,Z 575.625,A -85,B 0,C 180,E1 -21462.309,E2 -21462.309} C_VEL
LIN {X 0,Y 199.582,Z 575.622,A -85,B 0,C 180,E1 -21465.228,E2 -21465.228} C_VEL
LIN {X 0,Y 199.64,Z 575.617,A -85,B 0,C 180,E1 -21470.678,E2 -21470.678} C_VEL
LIN {X 0,Y 199.633,Z 575.615,A -85,B 0,C 180,E1 -21475.716,E2 -21475.716} C_VEL
LIN {X 0,Y 199.696,Z 575.605,A -85,B 0,C 180,E1 -21478.135,E2 -21478.135} C_VEL
LIN {X 0,Y 199.685,Z 575.612,A -85,B 0,C 180,E1 -21482.77,E2 -21482.77} C_VEL
LIN {X 0,Y 199.737,Z 575.601,A -85,B 0,C 180,E1 -21487.228,E2 -21487.228} C_VEL
LIN {X 0,Y 199.837,Z 575.59,A -85,B 0,C 180,E1 -21491.721,E2 -21491.721} C_VEL
LIN {X 0,Y 199.847,Z 575.585,A -85,B 0,C 180,E1 -21495.748,E2 -21495.748} C_VEL
LIN {X 0,Y 200.074,Z 575.561,A -85,B 0,C 180,E1 -21499.883,E2 -21499.883} C_VEL
LIN {X 0,Y 200.131,Z 575.553,A -85,B 0,C 180,E1 -21501.924,E2 -21501.924} C_VEL
LIN {X 0,Y 200.321,Z 575.53,A -85,B 0,C 180,E1 -21507.988,E2 -21507.988} C_VEL
LIN {X 0,Y 200.478,Z 575.51,A -85,B 0,C 180,E1 -21509.999,E2 -21509.999} C_VEL
LIN {X 0,Y 200.031,Z 575.564,A -85,B 0,C 180,E1 -21514.028,E2 -21514.028} C_VEL
LIN {X 0,Y 200.13,Z 575.554,A -85,B 0,C 180,E1 -21518.074,E2 -21518.074} C_VEL
LIN {X 0,Y 199.912,Z 575.577,A -85,B 0,C 180,E1 -21522.176,E2 -21522.176} C_VEL
LIN {X 0,Y 199.803,Z 575.595,A -85,B 0,C 180,E1 -21526.342,E2 -21526.342} C_VEL
LIN {X 0,Y 199.738,Z 575.599,A -85,B 0,C 180,E1 -21530.6,E2 -21530.6} C_VEL
LIN {X 0,Y 199.672,Z 575.612,A -85,B 0,C 180,E1 -21534.983,E2 -21534.983} C_VEL
LIN {X 0,Y 199.671,Z 575.61,A -85,B 0,C 180,E1 -21539.521,E2 -21539.521} C_VEL
LIN {X 0,Y 199.66,Z 575.613,A -85,B 0,C 180,E1 -21542.352,E2 -21542.352} C_VEL
LIN {X 0,Y 199.648,Z 575.614,A -85,B 0,C 180,E1 -21546.756,E2 -21546.756} C_VEL
LIN {X 0,Y 199.673,Z 575.612,A -85,B 0,C 180,E1 -21549.311,E2 -21549.311} C_VEL
LIN {X 0,Y 199.707,Z 575.607,A -85,B 0,C 180,E1 -21553.112,E2 -21553.112} C_VEL
LIN {X 0,Y 212.811,Z 612.368,A -85,B 0,C 180,E1 -21556.258,E2 -21556.258} C_VEL
LIN {X 0,Y 211.603,Z 644.179,A -85,B 0,C 180,E1 -21557.9,E2 -21557.9} C_VEL
LIN {X 0,Y 210.746,Z 658.068,A -85,B 0,C 180,E1 -21558.965,E2 -21558.965} C_VEL
LIN {X 0,Y 209.437,Z 672.855,A -85,B 0,C 180,E1 -21560.514,E2 -21560.514} C_VEL
LIN {X 0,Y 207.998,Z 685.661,A -85,B 0,C 180,E1 -21562.236,E2 -21562.236} C_VEL
LIN {X 0,Y 206.395,Z 698.119,A -85,B 0,C 180,E1 -21564.33,E2 -21564.33} C_VEL
LIN {X 0,Y 204.828,Z 709.586,A -85,B 0,C 180,E1 -21566.704,E2 -21566.704} C_VEL
LIN {X 0,Y 203.231,Z 720.77,A -85,B 0,C 180,E1 -21569.522,E2 -21569.522} C_VEL
LIN {X 0,Y 201.926,Z 730.555,A -85,B 0,C 180,E1 -21572.539,E2 -21572.539} C_VEL
LIN {X 0,Y 200.863,Z 739.267,A -85,B 0,C 180,E1 -21575.835,E2 -21575.835} C_VEL
LIN {X 0,Y 200.094,Z 746.996,A -85,B 0,C 180,E1 -21579.438,E2 -21579.438} C_VEL
LIN {X 0,Y 199.822,Z 752.544,A -85,B 0,C 180,E1 -21582.685,E2 -21582.685} C_VEL
LIN {X 0,Y 199.954,Z 756.758,A -85,B 0,C 180,E1 -21585.758,E2 -21585.758} C_VEL
LIN {X 0,Y 200.473,Z 760.223,A -85,B 0,C 180,E1 -21588.984,E2 -21588.984} C_VEL
LIN {X 0,Y 201.282,Z 762.624,A -85,B 0,C 180,E1 -21591.972,E2 -21591.972} C_VEL
LIN {X 0,Y 203.111,Z 764.588,A -85,B 0,C 180,E1 -21596.033,E2 -21596.033} C_VEL
LIN {X 0,Y 205.626,Z 765.136,A -85,B 0,C 180,E1 -21600.001,E2 -21600.001} C_VEL
LIN {X 0,Y 209.013,Z 764.22,A -85,B 0,C 180,E1 -21603.857,E2 -21603.857} C_VEL
LIN {X 0,Y 213.092,Z 761.847,A -85,B 0,C 180,E1 -21607.582,E2 -21607.582} C_VEL
LIN {X 0,Y 217.893,Z 757.976,A -85,B 0,C 180,E1 -21611.159,E2 -21611.159} C_VEL
LIN {X 0,Y 221.982,Z 754.007,A -85,B 0,C 180,E1 -21613.737,E2 -21613.737} C_VEL
LIN {X 0,Y 227.531,Z 747.761,A -85,B 0,C 180,E1 -21616.762,E2 -21616.762} C_VEL
LIN {X 0,Y 232.934,Z 740.637,A -85,B 0,C 180,E1 -21619.384,E2 -21619.384} C_VEL
LIN {X 0,Y 238.109,Z 732.769,A -85,B 0,C 180,E1 -21621.652,E2 -21621.652} C_VEL
LIN {X 0,Y 243.663,Z 723.212,A -85,B 0,C 180,E1 -21623.817,E2 -21623.817} C_VEL
LIN {X 0,Y 248.798,Z 712.677,A -85,B 0,C 180,E1 -21625.742,E2 -21625.742} C_VEL
LIN {X 0,Y 254.111,Z 699.802,A -85,B 0,C 180,E1 -21627.554,E2 -21627.554} C_VEL
LIN {X 0,Y 258.075,Z 687.687,A -85,B 0,C 180,E1 -21628.907,E2 -21628.907} C_VEL
LIN {X 0,Y 261.577,Z 673.899,A -85,B 0,C 180,E1 -21630.139,E2 -21630.139} C_VEL
LIN {X 0,Y 264.003,Z 660.663,A -85,B 0,C 180,E1 -21631.019,E2 -21631.019} C_VEL
LIN {X 0,Y 265.255,Z 651.71,A -85,B 0,C 180,E1 -21631.524,E2 -21631.524} C_VEL
LIN {X 0,Y 264.167,Z 649.094,A -85,B 0,C 180,E1 -21633.089,E2 -21633.089} C_VEL
LIN {X 0,Y 263.407,Z 646.831,A -85,B 0,C 180,E1 -21634.654,E2 -21634.654} C_VEL
LIN {X 0,Y 262.526,Z 645.693,A -85,B 0,C 180,E1 -21637.27,E2 -21637.27} C_VEL
LIN {X 0,Y 262.573,Z 645.93,A -85,B 0,C 180,E1 -21639.97,E2 -21639.97} C_VEL
LIN {X 0,Y 263.042,Z 646.919,A -85,B 0,C 180,E1 -21641.686,E2 -21641.686} C_VEL
LIN {X 0,Y 262.774,Z 650.615,A -85,B 0,C 180,E1 -21642.523,E2 -21642.523} C_VEL
LIN {X 0,Y 261.145,Z 664.504,A -85,B 0,C 180,E1 -21644.208,E2 -21644.208} C_VEL
LIN {X 0,Y 261.002,Z 665.807,A -85,B 0,C 180,E1 -21644.353,E2 -21644.353} C_VEL
LIN {X 0,Y 260.299,Z 671.271,A -85,B 0,C 180,E1 -21644.821,E2 -21644.821} C_VEL
LIN {X 0,Y 259.26,Z 677.044,A -85,B 0,C 180,E1 -21645.044,E2 -21645.044} C_VEL
LIN {X 0,Y 255.864,Z 690.81,A -85,B 0,C 180,E1 -21645.232,E2 -21645.232} C_VEL
LIN {X 0,Y 254.482,Z 696.315,A -85,B 0,C 180,E1 -21645.559,E2 -21645.559} C_VEL
LIN {X 0,Y 252.049,Z 705.865,A -85,B 0,C 180,E1 -21646.362,E2 -21646.362} C_VEL
LIN {X 0,Y 246.657,Z 720.968,A -85,B 0,C 180,E1 -21647.415,E2 -21647.415} C_VEL
LIN {X 0,Y 240.65,Z 734.741,A -85,B 0,C 180,E1 -21648.645,E2 -21648.645} C_VEL
LIN {X 0,Y 234.266,Z 747.372,A -85,B 0,C 180,E1 -21650.116,E2 -21650.116} C_VEL
LIN {X 0,Y 227.755,Z 758.918,A -85,B 0,C 180,E1 -21651.893,E2 -21651.893} C_VEL
LIN {X 0,Y 221.165,Z 769.467,A -85,B 0,C 180,E1 -21653.995,E2 -21653.995} C_VEL
LIN {X 0,Y 215.18,Z 778.426,A -85,B 0,C 180,E1 -21656.274,E2 -21656.274} C_VEL
LIN {X 0,Y 209.749,Z 786.01,A -85,B 0,C 180,E1 -21658.713,E2 -21658.713} C_VEL
LIN {X 0,Y 204.958,Z 792.474,A -85,B 0,C 180,E1 -21661.312,E2 -21661.312} C_VEL
LIN {X 0,Y 199.692,Z 799.514,A -85,B 0,C 180,E1 -21665.02,E2 -21665.02} C_VEL
LIN {X 0,Y 196.584,Z 803.701,A -85,B 0,C 180,E1 -21667.953,E2 -21667.953} C_VEL
LIN {X 0,Y 194.244,Z 807.067,A -85,B 0,C 180,E1 -21670.997,E2 -21670.997} C_VEL
LIN {X 0,Y 192.193,Z 810.282,A -85,B 0,C 180,E1 -21675.17,E2 -21675.17} C_VEL
LIN {X 0,Y 191.552,Z 812.113,A -85,B 0,C 180,E1 -21679.431,E2 -21679.431} C_VEL
LIN {X 0,Y 192.091,Z 812.512,A -85,B 0,C 180,E1 -21683.7,E2 -21683.7} C_VEL
LIN {X 0,Y 192.742,Z 812.126,A -85,B 0,C 180,E1 -21685.819,E2 -21685.819} C_VEL
LIN {X 0,Y 193.485,Z 811.315,A -85,B 0,C 180,E1 -21687.92,E2 -21687.92} C_VEL
LIN {X 0,Y 194.377,Z 810.093,A -85,B 0,C 180,E1 -21690.001,E2 -21690.001} C_VEL
LIN {X 0,Y 194.33,Z 809.681,A -85,B 0,C 180,E1 -21690.778,E2 -21690.778} C_VEL
LIN {X 0,Y 192.972,Z 811.668,A -85,B 0,C 180,E1 -21694.178,E2 -21694.178} C_VEL
LIN {X 0,Y 191.83,Z 812.659,A -85,B 0,C 180,E1 -21698.428,E2 -21698.428} C_VEL
LIN {X 0,Y 191.755,Z 812.259,A -85,B 0,C 180,E1 -21702.705,E2 -21702.705} C_VEL
LIN {X 0,Y 193.007,Z 810.571,A -85,B 0,C 180,E1 -21706.937,E2 -21706.937} C_VEL
LIN {X 0,Y 195.556,Z 807.624,A -85,B 0,C 180,E1 -21711.064,E2 -21711.064} C_VEL
LIN {X 0,Y 199.726,Z 803.442,A -85,B 0,C 180,E1 -21714.979,E2 -21714.979} C_VEL
LIN {X 0,Y 205.143,Z 797.964,A -85,B 0,C 180,E1 -21718.662,E2 -21718.662} C_VEL
LIN {X 0,Y 211.725,Z 791.104,A -85,B 0,C 180,E1 -21722.081,E2 -21722.081} C_VEL
LIN {X 0,Y 219.497,Z 782.752,A -85,B 0,C 180,E1 -21725.194,E2 -21725.194} C_VEL
LIN {X 0,Y 227.138,Z 774.074,A -85,B 0,C 180,E1 -21727.67,E2 -21727.67} C_VEL
LIN {X 0,Y 236.88,Z 762.344,A -85,B 0,C 180,E1 -21730.189,E2 -21730.189} C_VEL
LIN {X 0,Y 245.382,Z 751.161,A -85,B 0,C 180,E1 -21732,E2 -21732} C_VEL
LIN {X 0,Y 254.589,Z 737.814,A -85,B 0,C 180,E1 -21733.642,E2 -21733.642} C_VEL
LIN {X 0,Y 262.8,Z 724.61,A -85,B 0,C 180,E1 -21734.858,E2 -21734.858} C_VEL
LIN {X 0,Y 271.327,Z 708.981,A -85,B 0,C 180,E1 -21735.956,E2 -21735.956} C_VEL
LIN {X 0,Y 273.977,Z 703.494,A -85,B 0,C 180,E1 -21736.332,E2 -21736.332} C_VEL
LIN {X 0,Y 273.93,Z 703.419,A -85,B 0,C 180,E1 -21736.719,E2 -21736.719} C_VEL
LIN {X 0,Y 266.938,Z 715.928,A -85,B 0,C 180,E1 -21738.333,E2 -21738.333} C_VEL
LIN {X 0,Y 260.006,Z 726.483,A -85,B 0,C 180,E1 -21740.061,E2 -21740.061} C_VEL
LIN {X 0,Y 252.054,Z 736.822,A -85,B 0,C 180,E1 -21742.162,E2 -21742.162} C_VEL
LIN {X 0,Y 245.066,Z 744.766,A -85,B 0,C 180,E1 -21744.245,E2 -21744.245} C_VEL
LIN {X 0,Y 237.406,Z 752.386,A -85,B 0,C 180,E1 -21746.793,E2 -21746.793} C_VEL
LIN {X 0,Y 231.586,Z 757.386,A -85,B 0,C 180,E1 -21748.941,E2 -21748.941} C_VEL
LIN {X 0,Y 224.363,Z 762.758,A -85,B 0,C 180,E1 -21751.974,E2 -21751.974} C_VEL
LIN {X 0,Y 217.806,Z 766.73,A -85,B 0,C 180,E1 -21755.198,E2 -21755.198} C_VEL
LIN {X 0,Y 211.943,Z 769.458,A -85,B 0,C 180,E1 -21758.606,E2 -21758.606} C_VEL
LIN {X 0,Y 205.888,Z 771.131,A -85,B 0,C 180,E1 -21762.901,E2 -21762.901} C_VEL
LIN {X 0,Y 202.425,Z 771.298,A -85,B 0,C 180,E1 -21765.934,E2 -21765.934} C_VEL
LIN {X 0,Y 199.052,Z 770.422,A -85,B 0,C 180,E1 -21769.831,E2 -21769.831} C_VEL
LIN {X 0,Y 196.386,Z 768.398,A -85,B 0,C 180,E1 -21773.836,E2 -21773.836} C_VEL
LIN {X 0,Y 194.51,Z 765.176,A -85,B 0,C 180,E1 -21777.928,E2 -21777.928} C_VEL
LIN {X 0,Y 193.303,Z 760.696,A -85,B 0,C 180,E1 -21782.083,E2 -21782.083} C_VEL
LIN {X 0,Y 192.835,Z 754.813,A -85,B 0,C 180,E1 -21786.276,E2 -21786.276} C_VEL
LIN {X 0,Y 193,Z 748.07,A -85,B 0,C 180,E1 -21790.135,E2 -21790.135} C_VEL
LIN {X 0,Y 193.514,Z 740.626,A -85,B 0,C 180,E1 -21793.653,E2 -21793.653} C_VEL
LIN {X 0,Y 194.517,Z 731.25,A -85,B 0,C 180,E1 -21797.341,E2 -21797.341} C_VEL
LIN {X 0,Y 195.686,Z 721.57,A -85,B 0,C 180,E1 -21800.497,E2 -21800.497} C_VEL
LIN {X 0,Y 197.214,Z 710.081,A -85,B 0,C 180,E1 -21803.634,E2 -21803.634} C_VEL
LIN {X 0,Y 199.041,Z 697.481,A -85,B 0,C 180,E1 -21806.472,E2 -21806.472} C_VEL
LIN {X 0,Y 200.952,Z 683.058,A -85,B 0,C 180,E1 -21809.124,E2 -21809.124} C_VEL
LIN {X 0,Y 202.516,Z 670.022,A -85,B 0,C 180,E1 -21811.077,E2 -21811.077} C_VEL
LIN {X 0,Y 204.147,Z 654.162,A -85,B 0,C 180,E1 -21812.98,E2 -21812.98} C_VEL
LIN {X 0,Y 205.43,Z 638.006,A -85,B 0,C 180,E1 -21814.437,E2 -21814.437} C_VEL
LIN {X 0,Y 206.485,Z 617.079,A -85,B 0,C 180,E1 -21815.776,E2 -21815.776} C_VEL
LIN {X 0,Y 192.61,Z 576.491,A -85,B 0,C 180,E1 -21819.467,E2 -21819.467} C_VEL
LIN {X 0,Y 192.493,Z 576.507,A -85,B 0,C 180,E1 -21823.922,E2 -21823.922} C_VEL
LIN {X 0,Y 192.525,Z 576.499,A -85,B 0,C 180,E1 -21828.921,E2 -21828.921} C_VEL
LIN {X 0,Y 192.61,Z 576.491,A -85,B 0,C 180,E1 -21833.391,E2 -21833.391} C_VEL
LIN {X 0,Y 192.605,Z 576.487,A -85,B 0,C 180,E1 -21837.059,E2 -21837.059} C_VEL
LIN {X 0,Y 192.66,Z 576.485,A -85,B 0,C 180,E1 -21841.69,E2 -21841.69} C_VEL
LIN {X 0,Y 192.705,Z 576.477,A -85,B 0,C 180,E1 -21846.347,E2 -21846.347} C_VEL
LIN {X 0,Y 192.78,Z 576.47,A -85,B 0,C 180,E1 -21851.412,E2 -21851.412} C_VEL
LIN {X 0,Y 192.852,Z 576.461,A -85,B 0,C 180,E1 -21857.369,E2 -21857.369} C_VEL
LIN {X 0,Y 193.078,Z 576.432,A -85,B 0,C 180,E1 -21861.627,E2 -21861.627} C_VEL
LIN {X 0,Y 193.263,Z 576.41,A -85,B 0,C 180,E1 -21867.915,E2 -21867.915} C_VEL
LIN {X 0,Y 193.442,Z 576.387,A -85,B 0,C 180,E1 -21869.999,E2 -21869.999} C_VEL
LIN {X 0,Y 192.978,Z 576.442,A -85,B 0,C 180,E1 -21874.176,E2 -21874.176} C_VEL
LIN {X 0,Y 193.077,Z 576.433,A -85,B 0,C 180,E1 -21878.371,E2 -21878.371} C_VEL
LIN {X 0,Y 192.851,Z 576.457,A -85,B 0,C 180,E1 -21882.629,E2 -21882.629} C_VEL
LIN {X 0,Y 192.778,Z 576.469,A -85,B 0,C 180,E1 -21888.586,E2 -21888.586} C_VEL
LIN {X 0,Y 192.665,Z 576.484,A -85,B 0,C 180,E1 -21894.227,E2 -21894.227} C_VEL
LIN {X 0,Y 192.646,Z 576.484,A -85,B 0,C 180,E1 -21898.891,E2 -21898.891} C_VEL
LIN {X 0,Y 192.596,Z 576.493,A -85,B 0,C 180,E1 -21903.185,E2 -21903.185} C_VEL
LIN {X 0,Y 192.595,Z 576.494,A -85,B 0,C 180,E1 -21908.34,E2 -21908.34} C_VEL
LIN {X 0,Y 192.655,Z 576.487,A -85,B 0,C 180,E1 -21912.492,E2 -21912.492} C_VEL
LIN {X 0,Y 205.887,Z 613.433,A -85,B 0,C 180,E1 -21915.792,E2 -21915.792} C_VEL
LIN {X 0,Y 204.598,Z 645.485,A -85,B 0,C 180,E1 -21917.532,E2 -21917.532} C_VEL
LIN {X 0,Y 203.683,Z 660.072,A -85,B 0,C 180,E1 -21918.709,E2 -21918.709} C_VEL
LIN {X 0,Y 202.416,Z 673.799,A -85,B 0,C 180,E1 -21920.202,E2 -21920.202} C_VEL
LIN {X 0,Y 200.959,Z 686.42,A -85,B 0,C 180,E1 -21921.949,E2 -21921.949} C_VEL
LIN {X 0,Y 199.498,Z 697.51,A -85,B 0,C 180,E1 -21923.837,E2 -21923.837} C_VEL
LIN {X 0,Y 197.891,Z 709.341,A -85,B 0,C 180,E1 -21926.296,E2 -21926.296} C_VEL
LIN {X 0,Y 196.213,Z 720.966,A -85,B 0,C 180,E1 -21929.273,E2 -21929.273} C_VEL
LIN {X 0,Y 194.962,Z 729.924,A -85,B 0,C 180,E1 -21932.056,E2 -21932.056} C_VEL
LIN {X 0,Y 193.974,Z 737.63,A -85,B 0,C 180,E1 -21934.927,E2 -21934.927} C_VEL
LIN {X 0,Y 193.233,Z 744.776,A -85,B 0,C 180,E1 -21938.113,E2 -21938.113} C_VEL
LIN {X 0,Y 192.753,Z 752.201,A -85,B 0,C 180,E1 -21942.22,E2 -21942.22} C_VEL
LIN {X 0,Y 192.96,Z 757.852,A -85,B 0,C 180,E1 -21946.307,E2 -21946.307} C_VEL
LIN {X 0,Y 193.51,Z 761.269,A -85,B 0,C 180,E1 -21949.538,E2 -21949.538} C_VEL
LIN {X 0,Y 194.927,Z 764.429,A -85,B 0,C 180,E1 -21953.791,E2 -21953.791} C_VEL
LIN {X 0,Y 197.119,Z 766.143,A -85,B 0,C 180,E1 -21957.958,E2 -21957.958} C_VEL
LIN {X 0,Y 200.161,Z 766.353,A -85,B 0,C 180,E1 -21962.013,E2 -21962.013} C_VEL
LIN {X 0,Y 204.009,Z 765.159,A -85,B 0,C 180,E1 -21965.933,E2 -21965.933} C_VEL
LIN {X 0,Y 208.629,Z 762.538,A -85,B 0,C 180,E1 -21969.698,E2 -21969.698} C_VEL
LIN {X 0,Y 212.538,Z 759.572,A -85,B 0,C 180,E1 -21972.413,E2 -21972.413} C_VEL
LIN {X 0,Y 216.925,Z 755.652,A -85,B 0,C 180,E1 -21975.023,E2 -21975.023} C_VEL
LIN {X 0,Y 222.303,Z 750.126,A -85,B 0,C 180,E1 -21977.822,E2 -21977.822} C_VEL
LIN {X 0,Y 228.549,Z 742.553,A -85,B 0,C 180,E1 -21980.71,E2 -21980.71} C_VEL
LIN {X 0,Y 234.051,Z 734.869,A -85,B 0,C 180,E1 -21982.978,E2 -21982.978} C_VEL
LIN {X 0,Y 239.876,Z 725.453,A -85,B 0,C 180,E1 -21985.141,E2 -21985.141} C_VEL
LIN {X 0,Y 245.277,Z 715.323,A -85,B 0,C 180,E1 -21987.034,E2 -21987.034} C_VEL
LIN {X 0,Y 250.738,Z 702.997,A -85,B 0,C 180,E1 -21988.801,E2 -21988.801} C_VEL
LIN {X 0,Y 255.119,Z 690.993,A -85,B 0,C 180,E1 -21990.183,E2 -21990.183} C_VEL
LIN {X 0,Y 258.533,Z 678.887,A -85,B 0,C 180,E1 -21991.306,E2 -21991.306} C_VEL
LIN {X 0,Y 261.396,Z 665.624,A -85,B 0,C 180,E1 -21992.262,E2 -21992.262} C_VEL
